// Mitsubishi GX Works2 project: FX3U Rev12-22-jul-2025 1727   PLC: FX3U/FX3UC

PROGRAM 0_HOME
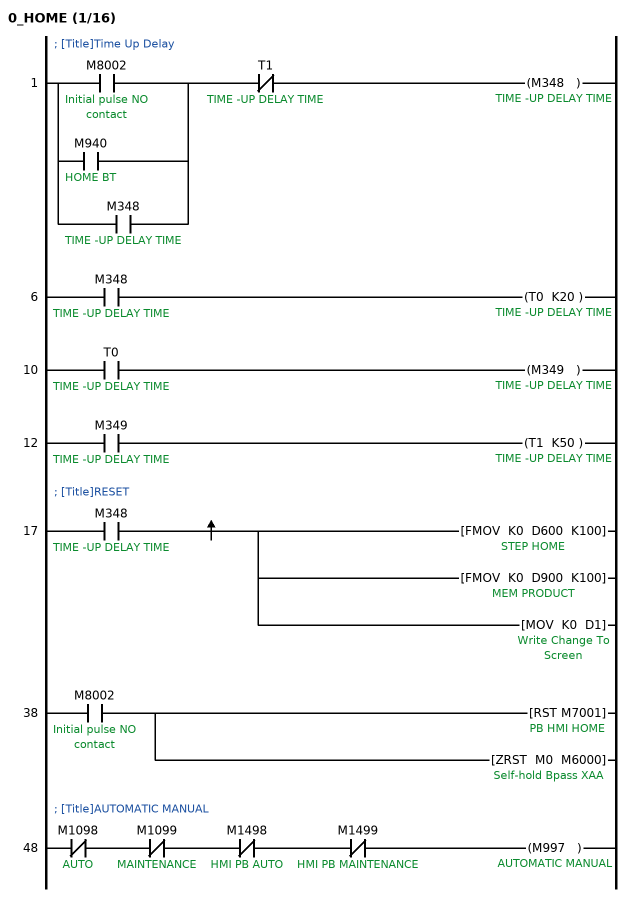
; [Title]Time Up Delay
1     LD      M8002  ; Initial pulse NO contact
      OR      M940  ; HOME BT
      OR      M348  ; TIME -UP DELAY TIME
      ANI     T1  ; TIME -UP DELAY TIME
      OUT     M348  ; TIME -UP DELAY TIME
6     LD      M348  ; TIME -UP DELAY TIME
      OUT     T0 K20  ; TIME -UP DELAY TIME
10    LD      T0  ; TIME -UP DELAY TIME
      OUT     M349  ; TIME -UP DELAY TIME
12    LD      M349  ; TIME -UP DELAY TIME
      OUT     T1 K50  ; TIME -UP DELAY TIME
; [Title]RESET
17    LD      M348  ; TIME -UP DELAY TIME
      MEP
      FMOV    K0 D600 K100  ; STEP HOME
      FMOV    K0 D900 K100  ; MEM PRODUCT
      MOV     K0 D1  ; Write Change To Screen
38    LD      M8002  ; Initial pulse NO contact
      RST     M7001  ; PB HMI HOME
      ZRST    M0 M6000  ; Self-hold Bpass XAA
; [Title]AUTOMATIC MANUAL
48    LDI     M1098  ; AUTO
      ANI     M1099  ; MAINTENANCE
      ANI     M1498  ; HMI PB AUTO
      ANI     M1499  ; HMI PB MAINTENANCE
      OUT     M997  ; AUTOMATIC MANUAL
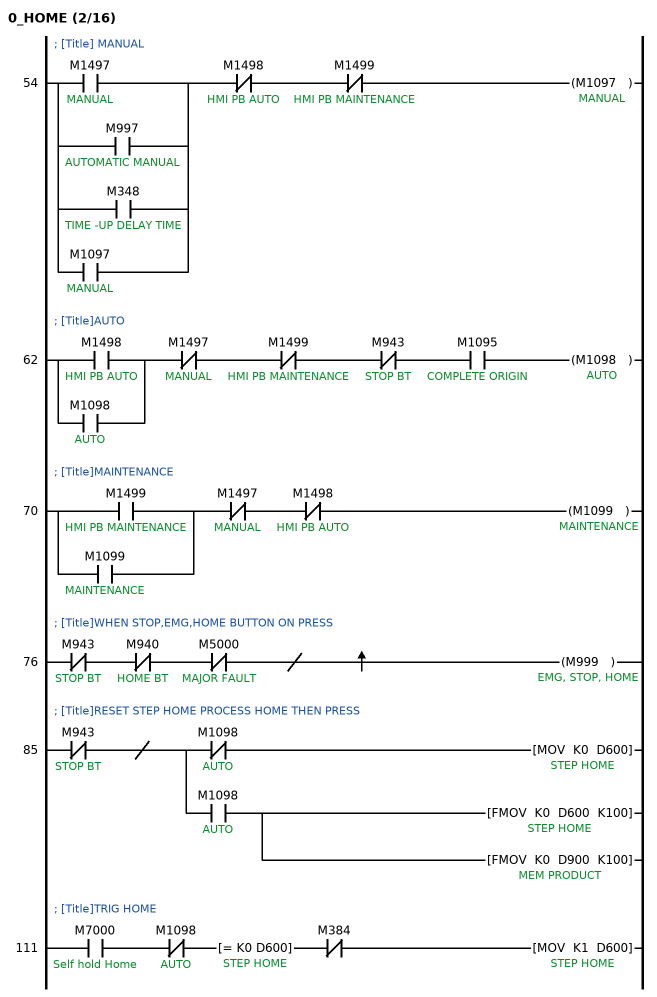
; [Title] MANUAL
54    LD      M1497  ; MANUAL
      OR      M997  ; AUTOMATIC MANUAL
      OR      M348  ; TIME -UP DELAY TIME
      OR      M1097  ; MANUAL
      ANI     M1498  ; HMI PB AUTO
      ANI     M1499  ; HMI PB MAINTENANCE
      OUT     M1097  ; MANUAL
; [Title]AUTO
62    LD      M1498  ; HMI PB AUTO
      OR      M1098  ; AUTO
      ANI     M1497  ; MANUAL
      ANI     M1499  ; HMI PB MAINTENANCE
      ANI     M943  ; STOP BT
      AND     M1095  ; COMPLETE ORIGIN
      OUT     M1098  ; AUTO
; [Title]MAINTENANCE
70    LD      M1499  ; HMI PB MAINTENANCE
      OR      M1099  ; MAINTENANCE
      ANI     M1497  ; MANUAL
      ANI     M1498  ; HMI PB AUTO
      OUT     M1099  ; MAINTENANCE
; [Title]WHEN STOP,EMG,HOME BUTTON ON PRESS
76    LDI     M943  ; STOP BT
      ANI     M940  ; HOME BT
      ANI     M5000  ; MAJOR FAULT
      INV
      MEP
      OUT     M999  ; EMG, STOP, HOME
; [Title]RESET STEP HOME PROCESS HOME THEN PRESS
85    LDI     M943  ; STOP BT
      INV
      MPS
      ANI     M1098  ; AUTO
      MOV     K0 D600
      MPP
      AND     M1098  ; AUTO
      FMOV    K0 D600 K100
      FMOV    K0 D900 K100
; [Title]TRIG HOME
111   LD      M7000  ; Self hold Home
      ANI     M1098  ; AUTO
      AND=    K0 D600  ; STEP HOME
      ANI     M384
      MOV     K1 D600
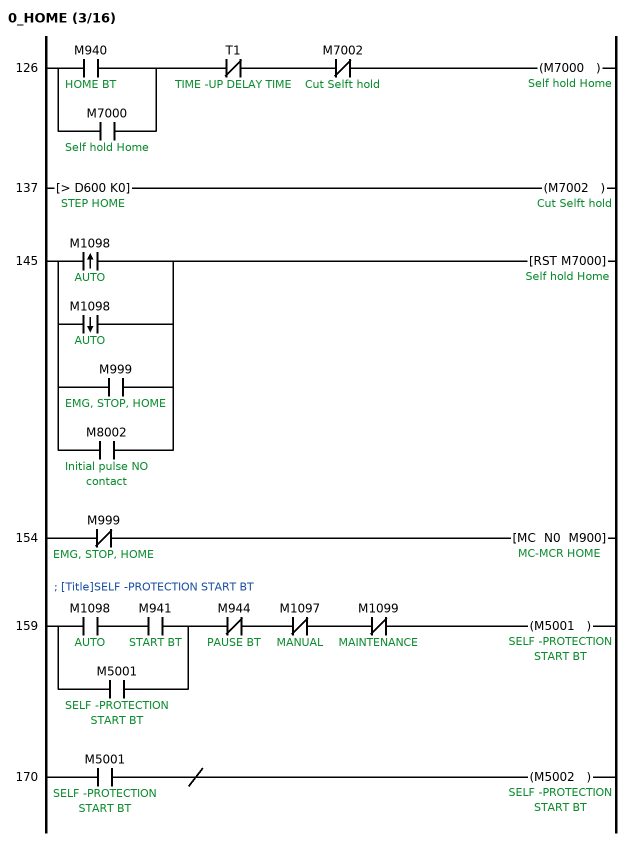
126   LD      M940  ; HOME BT
      OR      M7000  ; Self hold Home
      ANI     T1  ; TIME -UP DELAY TIME
      ANI     M7002  ; Cut Selft hold
      OUT     M7000  ; Self hold Home
137   LD>     D600 K0  ; STEP HOME
      OUT     M7002  ; Cut Selft hold
145   LDP     M1098  ; AUTO
      ORF     M1098  ; AUTO
      OR      M999  ; EMG, STOP, HOME
      OR      M8002  ; Initial pulse NO contact
      RST     M7000  ; Self hold Home
154   LDI     M999  ; EMG, STOP, HOME
      MC      N0 M900  ; MC-MCR HOME
; [Title]SELF -PROTECTION START BT
159   LD      M1098  ; AUTO
      AND     M941  ; START BT
      OR      M5001  ; SELF -PROTECTION START BT
      ANI     M944  ; PAUSE BT
      ANI     M1097  ; MANUAL
      ANI     M1099  ; MAINTENANCE
      OUT     M5001  ; SELF -PROTECTION START BT
170   LD      M5001  ; SELF -PROTECTION START BT
      INV
      OUT     M5002  ; SELF -PROTECTION START BT
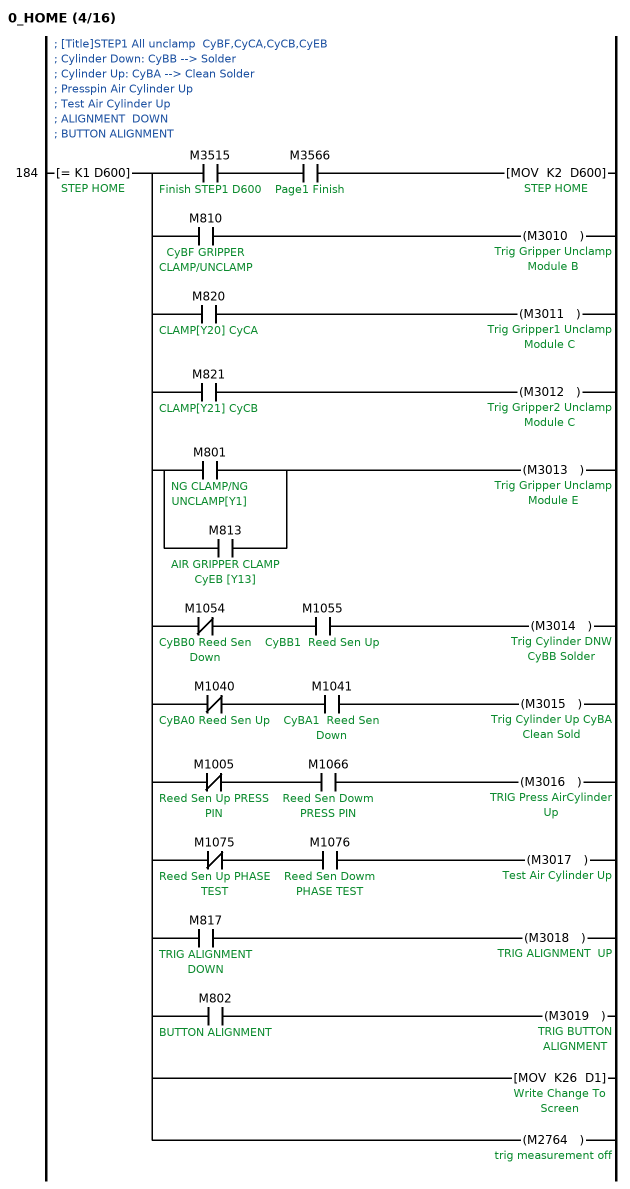
; [Title]STEP1 All unclamp  CyBF,CyCA,CyCB,CyEB
; Cylinder Down: CyBB --> Solder
; Cylinder Up: CyBA --> Clean Solder
; Presspin Air Cylinder Up
; Test Air Cylinder Up
; ALIGNMENT  DOWN
; BUTTON ALIGNMENT
184   LD=     K1 D600  ; STEP HOME
      MPS
      AND     M3515  ; Finish STEP1 D600
      AND     M3566  ; Page1 Finish
      MOV     K2 D600
      MRD
      AND     M810  ; CyBF GRIPPER CLAMP/UNCLAMP
      OUT     M3010  ; Trig Gripper Unclamp Module B
        [note] TRIG Gripper Unclamp Module B
      MRD
      AND     M820  ; CLAMP[Y20] CyCA
      OUT     M3011  ; Trig Gripper1 Unclamp Module C
        [note] TRIG Gripper1 Unclamp Module C
      MRD
      AND     M821  ; CLAMP[Y21] CyCB
      OUT     M3012  ; Trig Gripper2 Unclamp Module C
        [note] TRIG Gripper2 Unclamp Module C
      MRD
      LD      M801  ; NG CLAMP/NG UNCLAMP[Y1]
      OR      M813  ; AIR GRIPPER CLAMP CyEB [Y13]
      ANB
      OUT     M3013  ; Trig Gripper Unclamp Module E
        [note] TRIG Gripper Unclamp Module E
      MRD
      ANI     M1054  ; CyBB0 Reed Sen Down
      AND     M1055  ; CyBB1  Reed Sen Up
      OUT     M3014  ; Trig Cylinder DNW CyBB Solder
        [note] TRIG Cylinder DNW CyBB Solder
      MRD
      ANI     M1040  ; CyBA0 Reed Sen Up
      AND     M1041  ; CyBA1  Reed Sen Down
      OUT     M3015  ; Trig Cylinder Up CyBA Clean Sold
        [note] TRIG Cylinder Up CyBA Clean
      MRD
      ANI     M1005  ; Reed Sen Up PRESS PIN
      AND     M1066  ; Reed Sen Dowm PRESS PIN
      OUT     M3016  ; TRIG Press AirCylinder Up
        [note] TRIG Press AirCylinder Up
      MRD
      ANI     M1075  ; Reed Sen Up PHASE TEST
      AND     M1076  ; Reed Sen Dowm PHASE TEST
      OUT     M3017  ; Test Air Cylinder Up
        [note] TRIG Test Air Cylinder Up
      MRD
      AND     M817  ; TRIG ALIGNMENT  DOWN
      OUT     M3018  ; TRIG ALIGNMENT  UP
        [note] TRIG ALIGNMENT  UP
      MRD
      AND     M802  ; BUTTON ALIGNMENT
      OUT     M3019  ; TRIG BUTTON ALIGNMENT
        [note] TRIG BUTTON ALIGNMENT
      MPP
      MOV     K26 D1
      OUT     M2764  ; trig measurement off
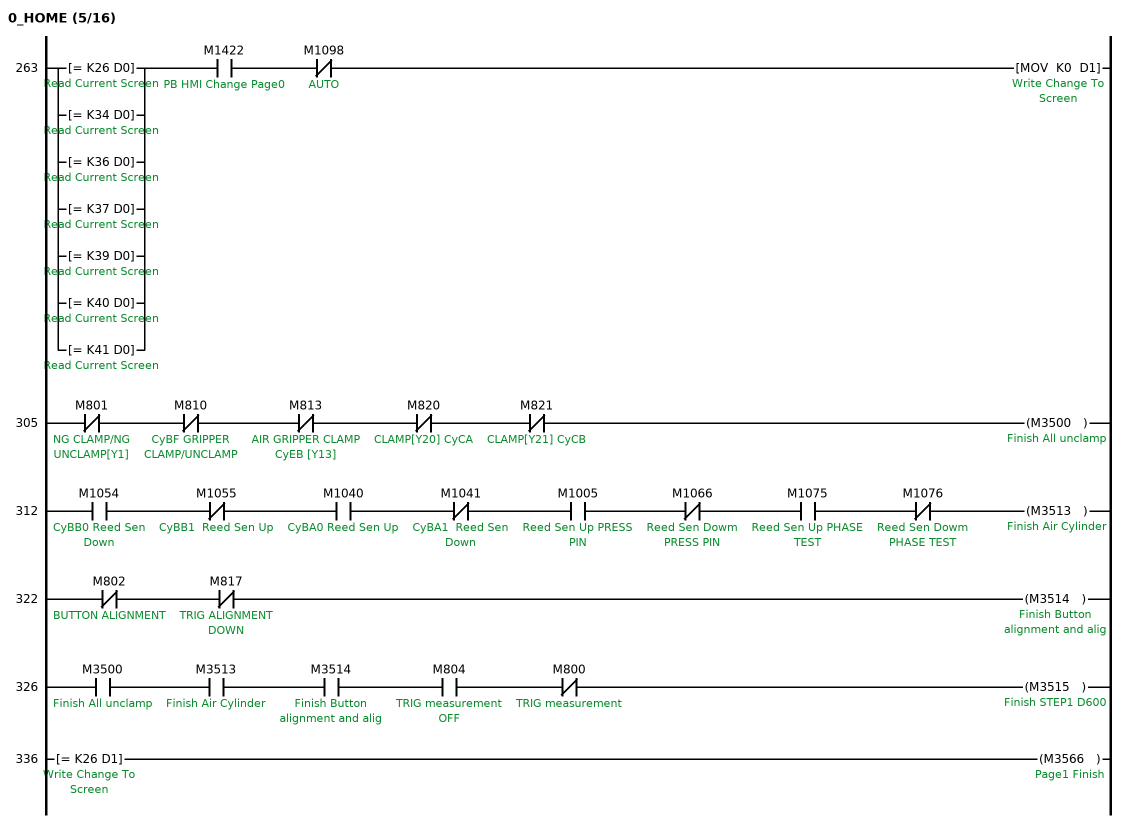
263   LD=     K26 D0  ; Read Current Screen
      OR=     K34 D0  ; Read Current Screen
      OR=     K36 D0  ; Read Current Screen
      OR=     K37 D0  ; Read Current Screen
      OR=     K39 D0  ; Read Current Screen
      OR=     K40 D0  ; Read Current Screen
      OR=     K41 D0  ; Read Current Screen
      AND     M1422  ; PB HMI Change Page0
      ANI     M1098  ; AUTO
      MOV     K0 D1
305   LDI     M801  ; NG CLAMP/NG UNCLAMP[Y1]
      ANI     M810  ; CyBF GRIPPER CLAMP/UNCLAMP
      ANI     M813  ; AIR GRIPPER CLAMP CyEB [Y13]
      ANI     M820  ; CLAMP[Y20] CyCA
      ANI     M821  ; CLAMP[Y21] CyCB
      OUT     M3500  ; Finish All unclamp
312   LD      M1054  ; CyBB0 Reed Sen Down
      ANI     M1055  ; CyBB1  Reed Sen Up
      AND     M1040  ; CyBA0 Reed Sen Up
      ANI     M1041  ; CyBA1  Reed Sen Down
      AND     M1005  ; Reed Sen Up PRESS PIN
      ANI     M1066  ; Reed Sen Dowm PRESS PIN
      AND     M1075  ; Reed Sen Up PHASE TEST
      ANI     M1076  ; Reed Sen Dowm PHASE TEST
      OUT     M3513  ; Finish Air Cylinder
322   LDI     M802  ; BUTTON ALIGNMENT
      ANI     M817  ; TRIG ALIGNMENT  DOWN
      OUT     M3514  ; Finish Button alignment and alig
326   LD      M3500  ; Finish All unclamp
      AND     M3513  ; Finish Air Cylinder
      AND     M3514  ; Finish Button alignment and alig
      AND     M804  ; TRIG measurement OFF
      ANI     M800  ; TRIG measurement
      OUT     M3515  ; Finish STEP1 D600
336   LD=     K26 D1  ; Write Change To Screen
      OUT     M3566  ; Page1 Finish
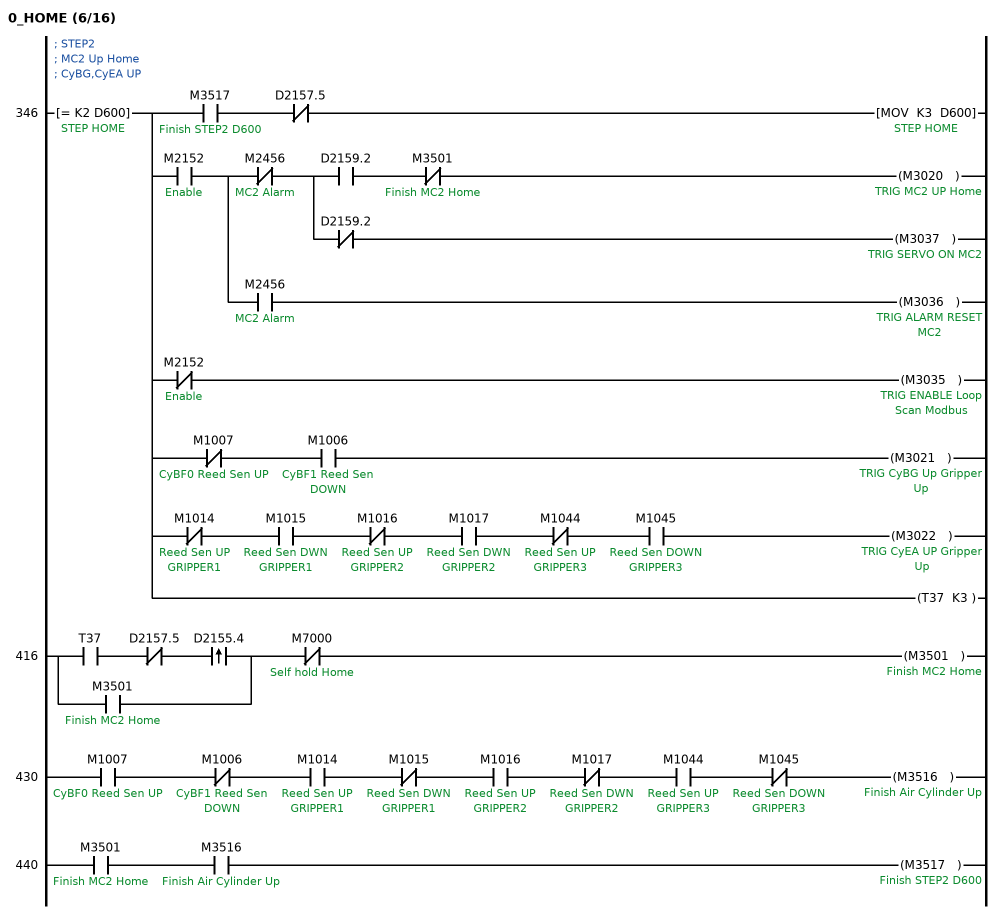
; STEP2
; MC2 Up Home
; CyBG,CyEA UP
346   LD=     K2 D600  ; STEP HOME
      MPS
      AND     M3517  ; Finish STEP2 D600
      ANI     D2157.5
      MOV     K3 D600
      MRD
      AND     M2152  ; Enable
      MPS
      ANI     M2456  ; MC2 Alarm
      MPS
      AND     D2159.2
      ANI     M3501  ; Finish MC2 Home
      OUT     M3020  ; TRIG MC2 UP Home
        [note] TRIG MC2 UP Home
      MPP
      ANI     D2159.2
      OUT     M3037  ; TRIG SERVO ON MC2
        [note] TRIG SERVO ON MC2
      MPP
      AND     M2456  ; MC2 Alarm
      OUT     M3036  ; TRIG ALARM RESET MC2
        [note] TRIG ALARM RESET MC2
      MRD
      ANI     M2152  ; Enable
      OUT     M3035  ; TRIG ENABLE Loop Scan Modbus
        [note] TRIG ENABLE Loop Scan Modbus
      MRD
      ANI     M1007  ; CyBF0 Reed Sen UP
      AND     M1006  ; CyBF1 Reed Sen DOWN
      OUT     M3021  ; TRIG CyBG Up Gripper Up
        [note] TRIG CyBG Up Gripper Up
      MRD
      ANI     M1014  ; Reed Sen UP GRIPPER1
      AND     M1015  ; Reed Sen DWN GRIPPER1
      ANI     M1016  ; Reed Sen UP GRIPPER2
      AND     M1017  ; Reed Sen DWN GRIPPER2
      ANI     M1044  ; Reed Sen UP GRIPPER3
      AND     M1045  ; Reed Sen DOWN GRIPPER3
      OUT     M3022  ; TRIG CyEA UP Gripper Up
        [note] TRIG CyEA UP Gripper Up
      MPP
      OUT     T37 K3
416   LD      T37
      ANI     D2157.5
      ANDP    D2155.4
      OR      M3501  ; Finish MC2 Home
      ANI     M7000  ; Self hold Home
      OUT     M3501  ; Finish MC2 Home
430   LD      M1007  ; CyBF0 Reed Sen UP
      ANI     M1006  ; CyBF1 Reed Sen DOWN
      AND     M1014  ; Reed Sen UP GRIPPER1
      ANI     M1015  ; Reed Sen DWN GRIPPER1
      AND     M1016  ; Reed Sen UP GRIPPER2
      ANI     M1017  ; Reed Sen DWN GRIPPER2
      AND     M1044  ; Reed Sen UP GRIPPER3
      ANI     M1045  ; Reed Sen DOWN GRIPPER3
      OUT     M3516  ; Finish Air Cylinder Up
440   LD      M3501  ; Finish MC2 Home
      AND     M3516  ; Finish Air Cylinder Up
      OUT     M3517  ; Finish STEP2 D600
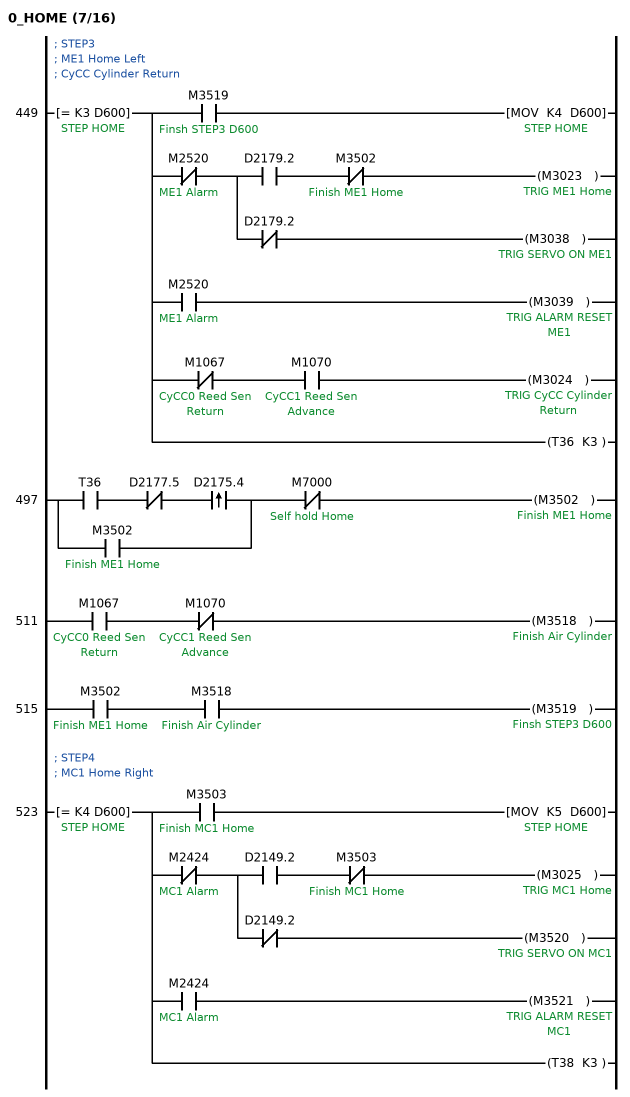
; STEP3
; ME1 Home Left
; CyCC Cylinder Return
449   LD=     K3 D600  ; STEP HOME
      MPS
      AND     M3519  ; Finsh STEP3 D600
      MOV     K4 D600
      MRD
      ANI     M2520  ; ME1 Alarm
      MPS
      AND     D2179.2
      ANI     M3502  ; Finish ME1 Home
      OUT     M3023  ; TRIG ME1 Home
        [note] TRIG ME1 Home
      MPP
      ANI     D2179.2
      OUT     M3038  ; TRIG SERVO ON ME1
        [note] TRIG SERVO ON ME1
      MRD
      AND     M2520  ; ME1 Alarm
      OUT     M3039  ; TRIG ALARM RESET ME1
        [note] TRIG ALARM RESET ME1
      MRD
      ANI     M1067  ; CyCC0 Reed Sen Return
      AND     M1070  ; CyCC1 Reed Sen  Advance
      OUT     M3024  ; TRIG CyCC Cylinder Return
        [note] TRIG CyCC Cylinder Return
      MPP
      OUT     T36 K3
497   LD      T36
      ANI     D2177.5
      ANDP    D2175.4
      OR      M3502  ; Finish ME1 Home
      ANI     M7000  ; Self hold Home
      OUT     M3502  ; Finish ME1 Home
511   LD      M1067  ; CyCC0 Reed Sen Return
      ANI     M1070  ; CyCC1 Reed Sen  Advance
      OUT     M3518  ; Finish Air Cylinder
515   LD      M3502  ; Finish ME1 Home
      AND     M3518  ; Finish Air Cylinder
      OUT     M3519  ; Finsh STEP3 D600
; STEP4
; MC1 Home Right
523   LD=     K4 D600  ; STEP HOME
      MPS
      AND     M3503  ; Finish MC1 Home
      MOV     K5 D600
      MRD
      ANI     M2424  ; MC1 Alarm
      MPS
      AND     D2149.2
      ANI     M3503  ; Finish MC1 Home
      OUT     M3025  ; TRIG MC1 Home
        [note] TRIG MC1 Home
      MPP
      ANI     D2149.2
      OUT     M3520  ; TRIG SERVO ON MC1
        [note] TRIG SERVO ON MC1
      MRD
      AND     M2424  ; MC1 Alarm
      OUT     M3521  ; TRIG ALARM RESET MC1
        [note] TRIG ALARM RESET MC1
      MPP
      OUT     T38 K3
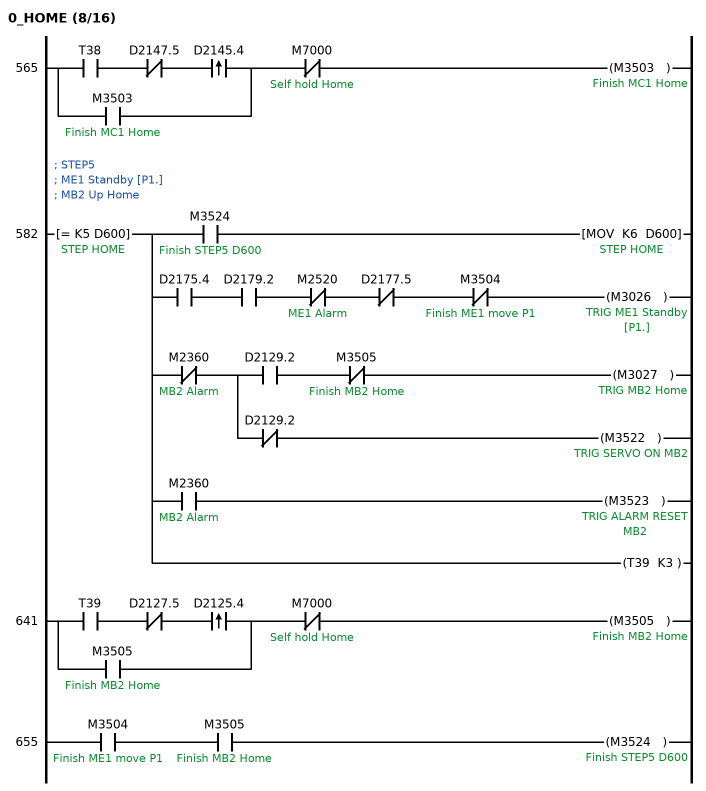
565   LD      T38
      ANI     D2147.5
      ANDP    D2145.4
      OR      M3503  ; Finish MC1 Home
      ANI     M7000  ; Self hold Home
      OUT     M3503  ; Finish MC1 Home
; STEP5
; ME1 Standby [P1.]
; MB2 Up Home
582   LD=     K5 D600  ; STEP HOME
      MPS
      AND     M3524  ; Finish STEP5 D600
      MOV     K6 D600
      MRD
      AND     D2175.4
      AND     D2179.2
      ANI     M2520  ; ME1 Alarm
      ANI     D2177.5
      ANI     M3504  ; Finish ME1 move P1
      OUT     M3026  ; TRIG ME1 Standby [P1.]
        [note] ME1 Standby [P1.]
      MRD
      ANI     M2360  ; MB2 Alarm
      MPS
      AND     D2129.2
      ANI     M3505  ; Finish MB2 Home
      OUT     M3027  ; TRIG MB2 Home
        [note] TRIG MB2 Home
      MPP
      ANI     D2129.2
      OUT     M3522  ; TRIG SERVO ON MB2
        [note] TRIG SERVO ON MB2
      MRD
      AND     M2360  ; MB2 Alarm
      OUT     M3523  ; TRIG ALARM RESET MB2
        [note] TRIG ALARM RESET MB2
      MPP
      OUT     T39 K3
641   LD      T39
      ANI     D2127.5
      ANDP    D2125.4
      OR      M3505  ; Finish MB2 Home
      ANI     M7000  ; Self hold Home
      OUT     M3505  ; Finish MB2 Home
655   LD      M3504  ; Finish ME1 move P1
      AND     M3505  ; Finish MB2 Home
      OUT     M3524  ; Finish STEP5 D600
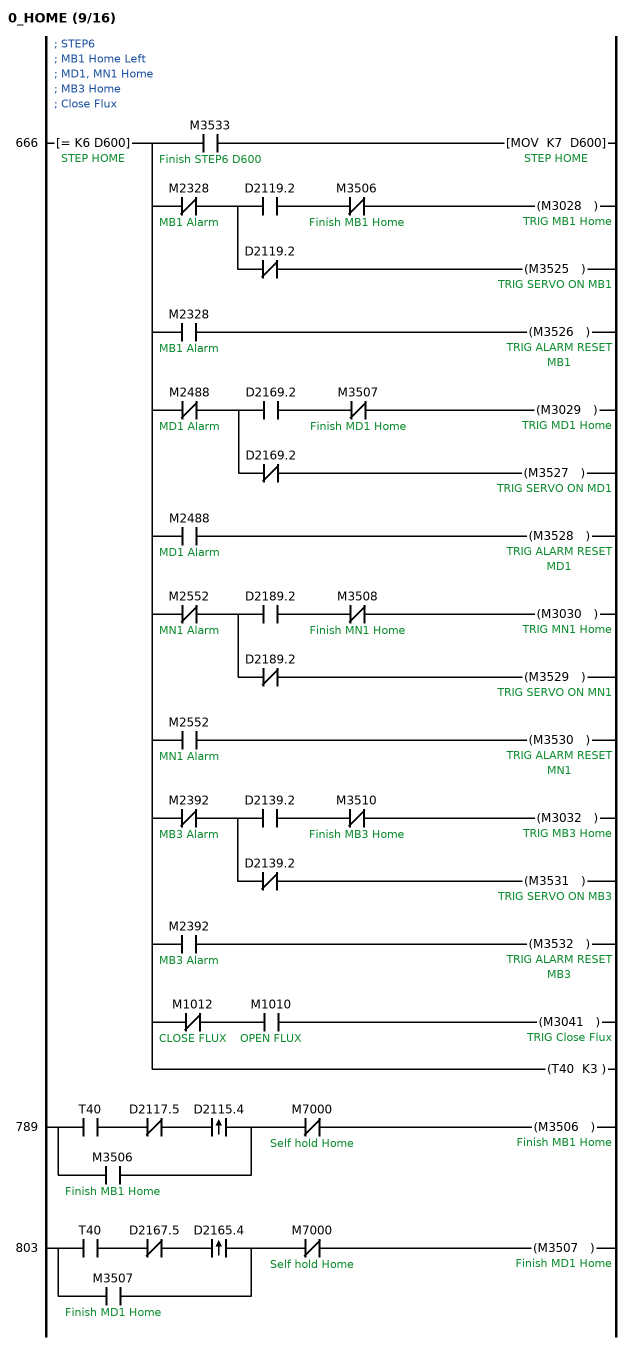
; STEP6
; MB1 Home Left
; MD1, MN1 Home
; MB3 Home
; Close Flux
666   LD=     K6 D600  ; STEP HOME
      MPS
      AND     M3533  ; Finish STEP6 D600
      MOV     K7 D600
      MRD
      ANI     M2328  ; MB1 Alarm
      MPS
      AND     D2119.2
      ANI     M3506  ; Finish MB1 Home
      OUT     M3028  ; TRIG MB1 Home
        [note] TRIG MB1 Home
      MPP
      ANI     D2119.2
      OUT     M3525  ; TRIG SERVO ON MB1
        [note] TRIG SERVO ON MB1
      MRD
      AND     M2328  ; MB1 Alarm
      OUT     M3526  ; TRIG ALARM RESET MB1
        [note] TRIG ALARM RESET MB1
      MRD
      ANI     M2488  ; MD1 Alarm
      MPS
      AND     D2169.2
      ANI     M3507  ; Finish MD1 Home
      OUT     M3029  ; TRIG MD1 Home
        [note] TRIG MD1 Home
      MPP
      ANI     D2169.2
      OUT     M3527  ; TRIG SERVO ON MD1
        [note] TRIG SERVO ON MD1
      MRD
      AND     M2488  ; MD1 Alarm
      OUT     M3528  ; TRIG ALARM RESET MD1
        [note] TRIG ALARM RESET MD1
      MRD
      ANI     M2552  ; MN1 Alarm
      MPS
      AND     D2189.2
      ANI     M3508  ; Finish MN1 Home
      OUT     M3030  ; TRIG MN1 Home
        [note] TRIG MN1 Home
      MPP
      ANI     D2189.2
      OUT     M3529  ; TRIG SERVO ON MN1
        [note] TRIG SERVO ON MN1
      MRD
      AND     M2552  ; MN1 Alarm
      OUT     M3530  ; TRIG ALARM RESET MN1
        [note] TRIG ALARM RESET MN1
      MRD
      ANI     M2392  ; MB3 Alarm
      MPS
      AND     D2139.2
      ANI     M3510  ; Finish MB3 Home
      OUT     M3032  ; TRIG MB3 Home
        [note] TRIG MB3 Home
      MPP
      ANI     D2139.2
      OUT     M3531  ; TRIG SERVO ON MB3
        [note] TRIG SERVO ON MB3
      MRD
      AND     M2392  ; MB3 Alarm
      OUT     M3532  ; TRIG ALARM RESET MB3
        [note] TRIG ALARM RESET MB3
      MRD
      ANI     M1012  ; CLOSE FLUX
      AND     M1010  ; OPEN FLUX
      OUT     M3041  ; TRIG Close Flux
        [note] TRIG Close Flux
      MPP
      OUT     T40 K3
789   LD      T40
      ANI     D2117.5
      ANDP    D2115.4
      OR      M3506  ; Finish MB1 Home
      ANI     M7000  ; Self hold Home
      OUT     M3506  ; Finish MB1 Home
803   LD      T40
      ANI     D2167.5
      ANDP    D2165.4
      OR      M3507  ; Finish MD1 Home
      ANI     M7000  ; Self hold Home
      OUT     M3507  ; Finish MD1 Home
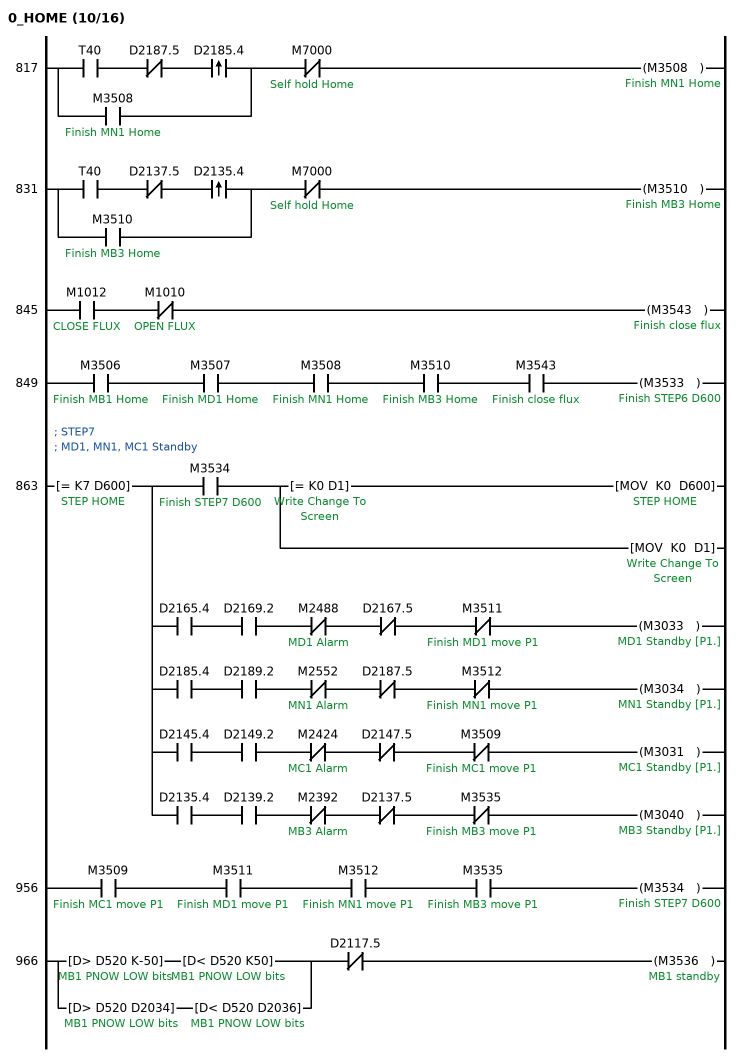
817   LD      T40
      ANI     D2187.5
      ANDP    D2185.4
      OR      M3508  ; Finish MN1 Home
      ANI     M7000  ; Self hold Home
      OUT     M3508  ; Finish MN1 Home
831   LD      T40
      ANI     D2137.5
      ANDP    D2135.4
      OR      M3510  ; Finish MB3 Home
      ANI     M7000  ; Self hold Home
      OUT     M3510  ; Finish MB3 Home
845   LD      M1012  ; CLOSE FLUX
      ANI     M1010  ; OPEN FLUX
      OUT     M3543  ; Finish close flux
849   LD      M3506  ; Finish MB1 Home
      AND     M3507  ; Finish MD1 Home
      AND     M3508  ; Finish MN1 Home
      AND     M3510  ; Finish MB3 Home
      AND     M3543  ; Finish close flux
      OUT     M3533  ; Finish STEP6 D600
; STEP7
; MD1, MN1, MC1 Standby
863   LD=     K7 D600  ; STEP HOME
      MPS
      AND     M3534  ; Finish STEP7 D600
      MPS
      AND=    K0 D1  ; Write Change To Screen
      MOV     K0 D600
      MPP
      MOV     K0 D1
      MRD
      AND     D2165.4
      AND     D2169.2
      ANI     M2488  ; MD1 Alarm
      ANI     D2167.5
      ANI     M3511  ; Finish MD1 move P1
      OUT     M3033  ; MD1 Standby [P1.]
        [note] MD1 Standby [P1.]
      MRD
      AND     D2185.4
      AND     D2189.2
      ANI     M2552  ; MN1 Alarm
      ANI     D2187.5
      ANI     M3512  ; Finish MN1 move P1
      OUT     M3034  ; MN1 Standby [P1.]
        [note] MN1 Standby [P1.]
      MRD
      AND     D2145.4
      AND     D2149.2
      ANI     M2424  ; MC1 Alarm
      ANI     D2147.5
      ANI     M3509  ; Finish MC1 move P1
      OUT     M3031  ; MC1 Standby [P1.]
        [note] MC1 Standby [P1.]
      MPP
      AND     D2135.4
      AND     D2139.2
      ANI     M2392  ; MB3 Alarm
      ANI     D2137.5
      ANI     M3535  ; Finish MB3 move P1
      OUT     M3040  ; MB3 Standby [P1.]
        [note] MB3 Standby [P1.]
956   LD      M3509  ; Finish MC1 move P1
      AND     M3511  ; Finish MD1 move P1
      AND     M3512  ; Finish MN1 move P1
      AND     M3535  ; Finish MB3 move P1
      OUT     M3534  ; Finish STEP7 D600
966   LDD>    D520 K-50  ; MB1 PNOW LOW bits
      ANDD<   D520 K50  ; MB1 PNOW LOW bits
      LDD>    D520 D2034  ; MB1 PNOW LOW bits
      ANDD<   D520 D2036  ; MB1 PNOW LOW bits
      ORB
      ANI     D2117.5
      OUT     M3536  ; MB1 standby
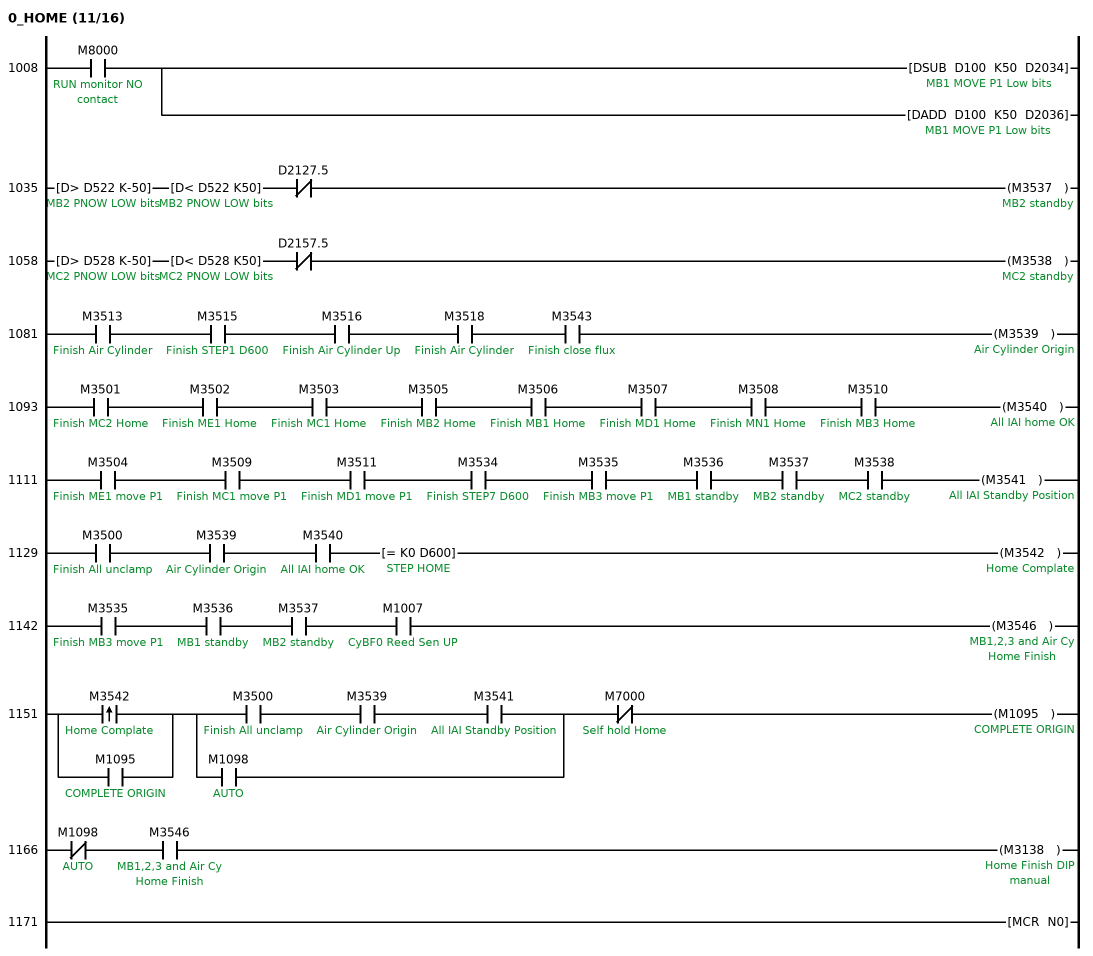
1008  LD      M8000  ; RUN monitor NO contact
      DSUB    D100 K50 D2034  ; MB1 MOVE P1 Low bits
      DADD    D100 K50 D2036
1035  LDD>    D522 K-50  ; MB2 PNOW LOW bits
      ANDD<   D522 K50  ; MB2 PNOW LOW bits
      ANI     D2127.5
      OUT     M3537  ; MB2 standby
1058  LDD>    D528 K-50  ; MC2 PNOW LOW bits
      ANDD<   D528 K50  ; MC2 PNOW LOW bits
      ANI     D2157.5
      OUT     M3538  ; MC2 standby
1081  LD      M3513  ; Finish Air Cylinder
      AND     M3515  ; Finish STEP1 D600
      AND     M3516  ; Finish Air Cylinder Up
      AND     M3518  ; Finish Air Cylinder
      AND     M3543  ; Finish close flux
      OUT     M3539  ; Air Cylinder Origin
1093  LD      M3501  ; Finish MC2 Home
      AND     M3502  ; Finish ME1 Home
      AND     M3503  ; Finish MC1 Home
      AND     M3505  ; Finish MB2 Home
      AND     M3506  ; Finish MB1 Home
      AND     M3507  ; Finish MD1 Home
      AND     M3508  ; Finish MN1 Home
      AND     M3510  ; Finish MB3 Home
      OUT     M3540  ; All IAI home OK
1111  LD      M3504  ; Finish ME1 move P1
      AND     M3509  ; Finish MC1 move P1
      AND     M3511  ; Finish MD1 move P1
      AND     M3534  ; Finish STEP7 D600
      AND     M3535  ; Finish MB3 move P1
      AND     M3536  ; MB1 standby
      AND     M3537  ; MB2 standby
      AND     M3538  ; MC2 standby
      OUT     M3541  ; All IAI Standby Position
1129  LD      M3500  ; Finish All unclamp
      AND     M3539  ; Air Cylinder Origin
      AND     M3540  ; All IAI home OK
      AND=    K0 D600  ; STEP HOME
      OUT     M3542  ; Home Complate
1142  LD      M3535  ; Finish MB3 move P1
      AND     M3536  ; MB1 standby
      AND     M3537  ; MB2 standby
      AND     M1007  ; CyBF0 Reed Sen UP
      OUT     M3546  ; MB1,2,3 and Air Cy Home Finish
1151  LDP     M3542  ; Home Complate
      OR      M1095  ; COMPLETE ORIGIN
      LD      M3500  ; Finish All unclamp
      AND     M3539  ; Air Cylinder Origin
      AND     M3541  ; All IAI Standby Position
      OR      M1098  ; AUTO
      ANB
      ANI     M7000  ; Self hold Home
      OUT     M1095  ; COMPLETE ORIGIN
1166  LDI     M1098  ; AUTO
      AND     M3546  ; MB1,2,3 and Air Cy Home Finish
      OUT     M3138  ; Home Finish DIP manual
1171  MCR     N0
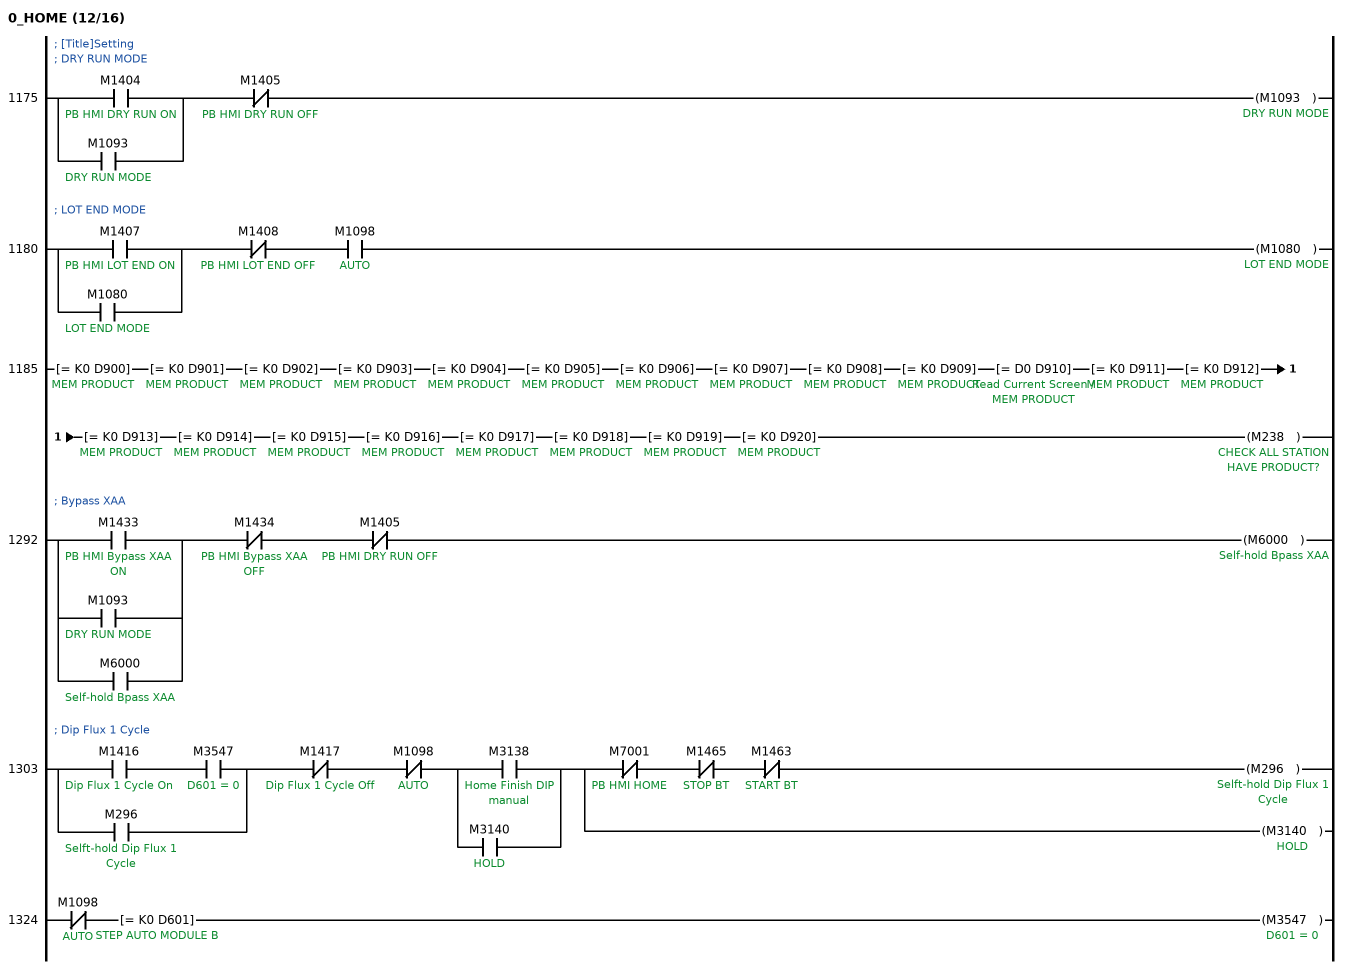
; [Title]Setting
; DRY RUN MODE
1175  LD      M1404  ; PB HMI DRY RUN ON
      OR      M1093  ; DRY RUN MODE
      ANI     M1405  ; PB HMI DRY RUN OFF
      OUT     M1093  ; DRY RUN MODE
; LOT END MODE
1180  LD      M1407  ; PB HMI LOT END ON
      OR      M1080  ; LOT END MODE
      ANI     M1408  ; PB HMI LOT END OFF
      AND     M1098  ; AUTO
      OUT     M1080  ; LOT END MODE
1185  LD=     K0 D900  ; MEM PRODUCT
      AND=    K0 D901  ; MEM PRODUCT
      AND=    K0 D902  ; MEM PRODUCT
      AND=    K0 D903  ; MEM PRODUCT
      AND=    K0 D904  ; MEM PRODUCT
      AND=    K0 D905  ; MEM PRODUCT
      AND=    K0 D906  ; MEM PRODUCT
      AND=    K0 D907  ; MEM PRODUCT
      AND=    K0 D908  ; MEM PRODUCT
      AND=    K0 D909  ; MEM PRODUCT
      AND=    D0 D910  ; Read Current Screen / MEM PRODUCT
      AND=    K0 D911  ; MEM PRODUCT
      AND=    K0 D912  ; MEM PRODUCT
      AND=    K0 D913  ; MEM PRODUCT
      AND=    K0 D914  ; MEM PRODUCT
      AND=    K0 D915  ; MEM PRODUCT
      AND=    K0 D916  ; MEM PRODUCT
      AND=    K0 D917  ; MEM PRODUCT
      AND=    K0 D918  ; MEM PRODUCT
      AND=    K0 D919  ; MEM PRODUCT
      AND=    K0 D920  ; MEM PRODUCT
      OUT     M238  ; CHECK ALL STATION HAVE PRODUCT?
; Bypass XAA
1292  LD      M1433  ; PB HMI Bypass XAA ON
      OR      M1093  ; DRY RUN MODE
      OR      M6000  ; Self-hold Bpass XAA
      ANI     M1434  ; PB HMI Bypass XAA OFF
      ANI     M1405  ; PB HMI DRY RUN OFF
      OUT     M6000  ; Self-hold Bpass XAA
; Dip Flux 1 Cycle
1303  LD      M1416  ; Dip Flux 1 Cycle On
      AND     M3547  ; D601 = 0
      OR      M296  ; Selft-hold Dip Flux 1 Cycle
      ANI     M1417  ; Dip Flux 1 Cycle Off
      ANI     M1098  ; AUTO
      LD      M3138  ; Home Finish DIP manual
      OR      M3140  ; HOLD
      ANB
      MPS
      ANI     M7001  ; PB HMI HOME
      ANI     M1465  ; STOP BT
      ANI     M1463  ; START BT
      OUT     M296  ; Selft-hold Dip Flux 1 Cycle
      MPP
      OUT     M3140  ; HOLD
1324  LDI     M1098  ; AUTO
      AND=    K0 D601  ; STEP AUTO MODULE B
      OUT     M3547  ; D601 = 0
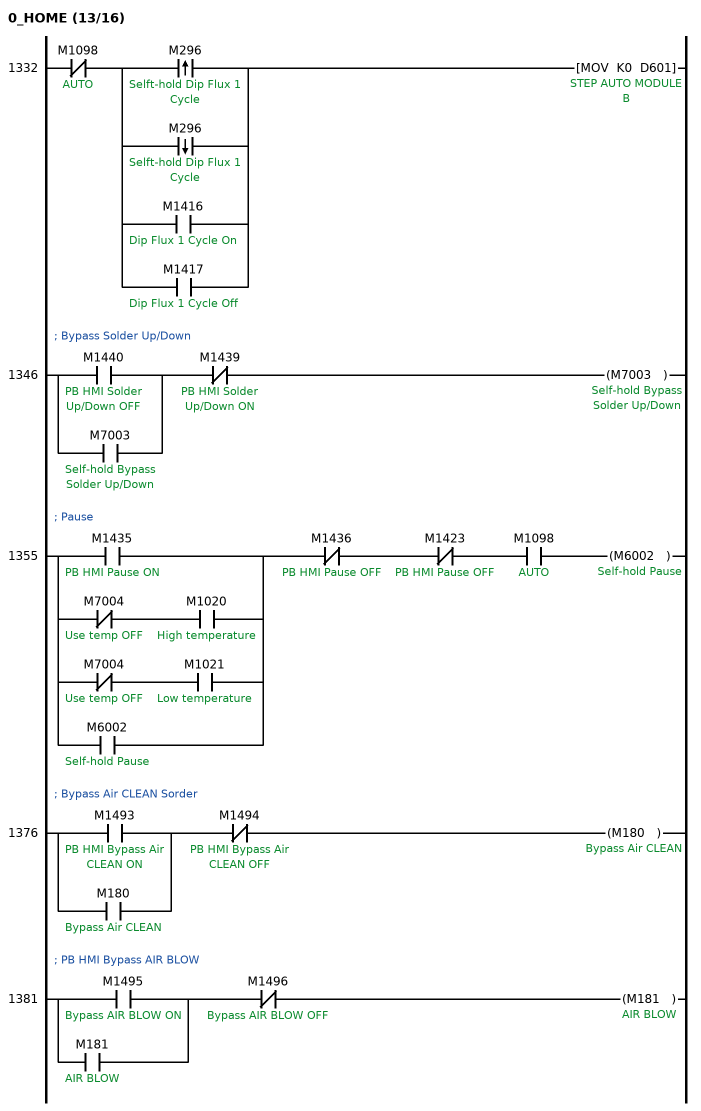
1332  LDI     M1098  ; AUTO
      LDP     M296  ; Selft-hold Dip Flux 1 Cycle
      ORF     M296  ; Selft-hold Dip Flux 1 Cycle
      OR      M1416  ; Dip Flux 1 Cycle On
      OR      M1417  ; Dip Flux 1 Cycle Off
      ANB
      MOV     K0 D601
; Bypass Solder Up/Down
1346  LD      M1440  ; PB HMI Solder Up/Down OFF
      OR      M7003  ; Self-hold Bypass Solder Up/Down
      ANI     M1439  ; PB HMI Solder Up/Down ON
      OUT     M7003  ; Self-hold Bypass Solder Up/Down
; Pause
1355  LD      M1435  ; PB HMI Pause ON
      LDI     M7004  ; Use temp OFF
      AND     M1020  ; High temperature
      ORB
      LDI     M7004  ; Use temp OFF
      AND     M1021  ; Low temperature
      ORB
      OR      M6002  ; Self-hold Pause
      ANI     M1436  ; PB HMI Pause OFF
      ANI     M1423  ; PB HMI Pause OFF
      AND     M1098  ; AUTO
      OUT     M6002  ; Self-hold Pause
; Bypass Air CLEAN Sorder
1376  LD      M1493  ; PB HMI Bypass Air CLEAN ON
      OR      M180  ; Bypass Air CLEAN
      ANI     M1494  ; PB HMI Bypass Air CLEAN OFF
      OUT     M180  ; Bypass Air CLEAN
; PB HMI Bypass AIR BLOW
1381  LD      M1495  ; Bypass AIR BLOW ON
      OR      M181  ; AIR BLOW
      ANI     M1496  ; Bypass AIR BLOW OFF
      OUT     M181  ; AIR BLOW
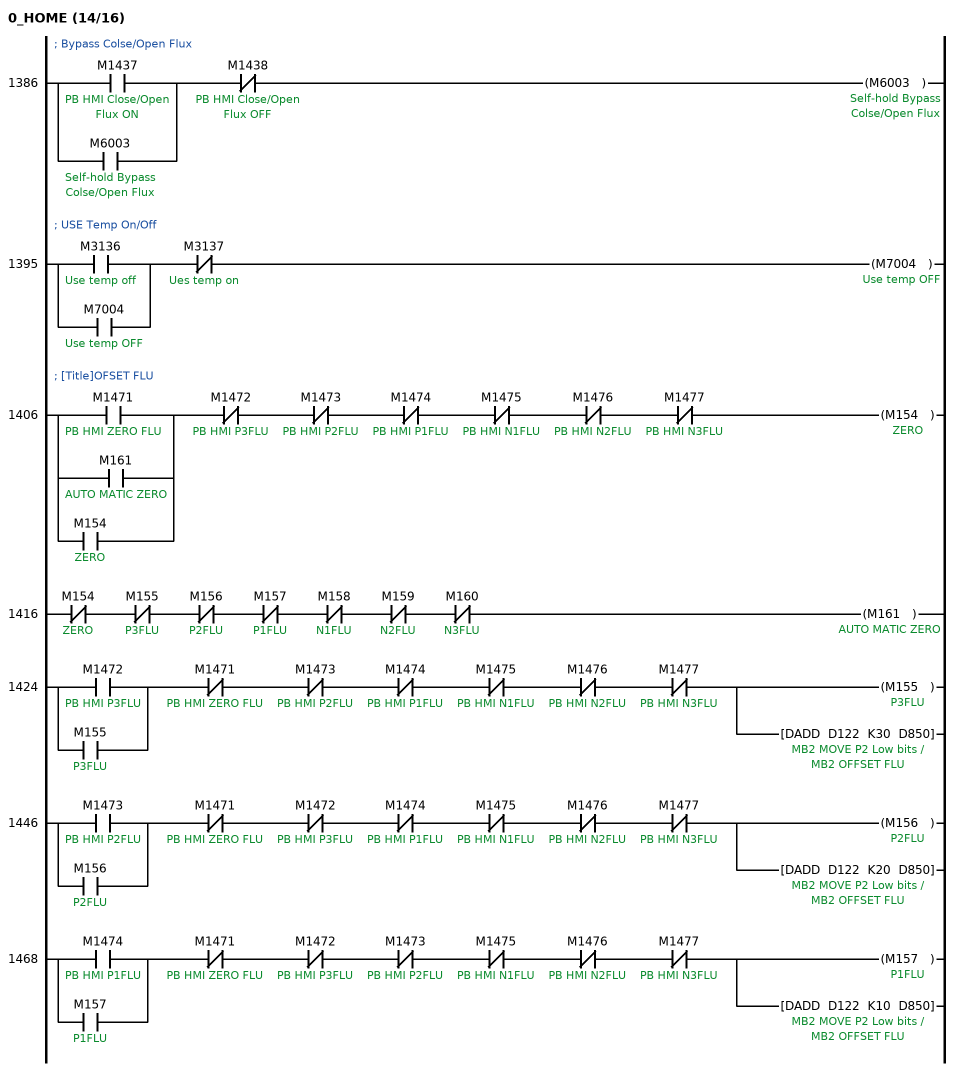
; Bypass Colse/Open Flux
1386  LD      M1437  ; PB HMI Close/Open Flux ON
      OR      M6003  ; Self-hold Bypass Colse/Open Flux
      ANI     M1438  ; PB HMI Close/Open Flux OFF
      OUT     M6003  ; Self-hold Bypass Colse/Open Flux
; USE Temp On/Off
1395  LD      M3136  ; Use temp off
      OR      M7004  ; Use temp OFF
      ANI     M3137  ; Ues temp on
      OUT     M7004  ; Use temp OFF
; [Title]OFSET FLU
1406  LD      M1471  ; PB HMI ZERO FLU
      OR      M161  ; AUTO MATIC ZERO
      OR      M154  ; ZERO
      ANI     M1472  ; PB HMI P3FLU
      ANI     M1473  ; PB HMI P2FLU
      ANI     M1474  ; PB HMI P1FLU
      ANI     M1475  ; PB HMI N1FLU
      ANI     M1476  ; PB HMI N2FLU
      ANI     M1477  ; PB HMI N3FLU
      OUT     M154  ; ZERO
1416  LDI     M154  ; ZERO
      ANI     M155  ; P3FLU
      ANI     M156  ; P2FLU
      ANI     M157  ; P1FLU
      ANI     M158  ; N1FLU
      ANI     M159  ; N2FLU
      ANI     M160  ; N3FLU
      OUT     M161  ; AUTO MATIC ZERO
1424  LD      M1472  ; PB HMI P3FLU
      OR      M155  ; P3FLU
      ANI     M1471  ; PB HMI ZERO FLU
      ANI     M1473  ; PB HMI P2FLU
      ANI     M1474  ; PB HMI P1FLU
      ANI     M1475  ; PB HMI N1FLU
      ANI     M1476  ; PB HMI N2FLU
      ANI     M1477  ; PB HMI N3FLU
      OUT     M155  ; P3FLU
      DADD    D122 K30 D850  ; MB2 MOVE P2 Low bits / MB2 OFFSET FLU
1446  LD      M1473  ; PB HMI P2FLU
      OR      M156  ; P2FLU
      ANI     M1471  ; PB HMI ZERO FLU
      ANI     M1472  ; PB HMI P3FLU
      ANI     M1474  ; PB HMI P1FLU
      ANI     M1475  ; PB HMI N1FLU
      ANI     M1476  ; PB HMI N2FLU
      ANI     M1477  ; PB HMI N3FLU
      OUT     M156  ; P2FLU
      DADD    D122 K20 D850
1468  LD      M1474  ; PB HMI P1FLU
      OR      M157  ; P1FLU
      ANI     M1471  ; PB HMI ZERO FLU
      ANI     M1472  ; PB HMI P3FLU
      ANI     M1473  ; PB HMI P2FLU
      ANI     M1475  ; PB HMI N1FLU
      ANI     M1476  ; PB HMI N2FLU
      ANI     M1477  ; PB HMI N3FLU
      OUT     M157  ; P1FLU
      DADD    D122 K10 D850
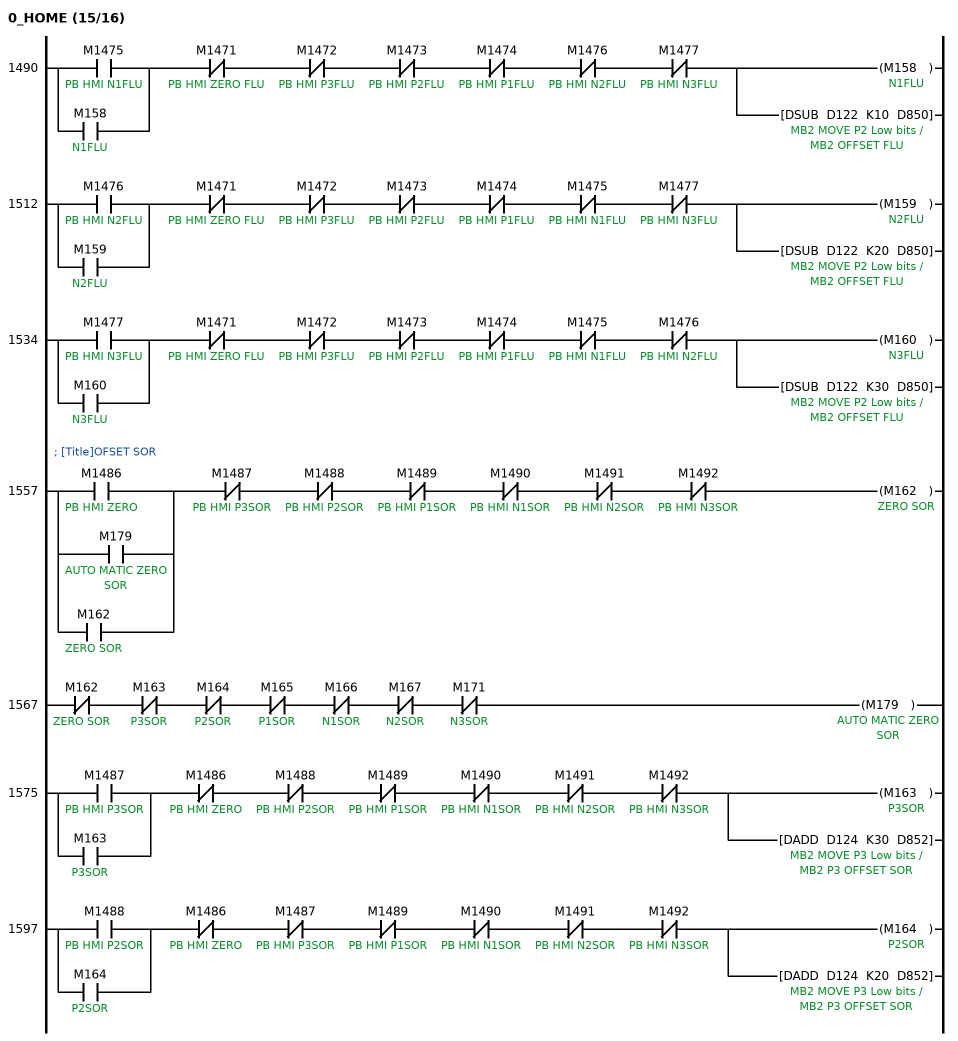
1490  LD      M1475  ; PB HMI N1FLU
      OR      M158  ; N1FLU
      ANI     M1471  ; PB HMI ZERO FLU
      ANI     M1472  ; PB HMI P3FLU
      ANI     M1473  ; PB HMI P2FLU
      ANI     M1474  ; PB HMI P1FLU
      ANI     M1476  ; PB HMI N2FLU
      ANI     M1477  ; PB HMI N3FLU
      OUT     M158  ; N1FLU
      DSUB    D122 K10 D850
1512  LD      M1476  ; PB HMI N2FLU
      OR      M159  ; N2FLU
      ANI     M1471  ; PB HMI ZERO FLU
      ANI     M1472  ; PB HMI P3FLU
      ANI     M1473  ; PB HMI P2FLU
      ANI     M1474  ; PB HMI P1FLU
      ANI     M1475  ; PB HMI N1FLU
      ANI     M1477  ; PB HMI N3FLU
      OUT     M159  ; N2FLU
      DSUB    D122 K20 D850
1534  LD      M1477  ; PB HMI N3FLU
      OR      M160  ; N3FLU
      ANI     M1471  ; PB HMI ZERO FLU
      ANI     M1472  ; PB HMI P3FLU
      ANI     M1473  ; PB HMI P2FLU
      ANI     M1474  ; PB HMI P1FLU
      ANI     M1475  ; PB HMI N1FLU
      ANI     M1476  ; PB HMI N2FLU
      OUT     M160  ; N3FLU
      DSUB    D122 K30 D850
; [Title]OFSET SOR
1557  LD      M1486  ; PB HMI ZERO
      OR      M179  ; AUTO MATIC ZERO SOR
      OR      M162  ; ZERO SOR
      ANI     M1487  ; PB HMI P3SOR
      ANI     M1488  ; PB HMI P2SOR
      ANI     M1489  ; PB HMI P1SOR
      ANI     M1490  ; PB HMI N1SOR
      ANI     M1491  ; PB HMI N2SOR
      ANI     M1492  ; PB HMI N3SOR
      OUT     M162  ; ZERO SOR
1567  LDI     M162  ; ZERO SOR
      ANI     M163  ; P3SOR
      ANI     M164  ; P2SOR
      ANI     M165  ; P1SOR
      ANI     M166  ; N1SOR
      ANI     M167  ; N2SOR
      ANI     M171  ; N3SOR
      OUT     M179  ; AUTO MATIC ZERO SOR
1575  LD      M1487  ; PB HMI P3SOR
      OR      M163  ; P3SOR
      ANI     M1486  ; PB HMI ZERO
      ANI     M1488  ; PB HMI P2SOR
      ANI     M1489  ; PB HMI P1SOR
      ANI     M1490  ; PB HMI N1SOR
      ANI     M1491  ; PB HMI N2SOR
      ANI     M1492  ; PB HMI N3SOR
      OUT     M163  ; P3SOR
      DADD    D124 K30 D852  ; MB2 MOVE P3 Low bits / MB2 P3 OFFSET SOR
1597  LD      M1488  ; PB HMI P2SOR
      OR      M164  ; P2SOR
      ANI     M1486  ; PB HMI ZERO
      ANI     M1487  ; PB HMI P3SOR
      ANI     M1489  ; PB HMI P1SOR
      ANI     M1490  ; PB HMI N1SOR
      ANI     M1491  ; PB HMI N2SOR
      ANI     M1492  ; PB HMI N3SOR
      OUT     M164  ; P2SOR
      DADD    D124 K20 D852
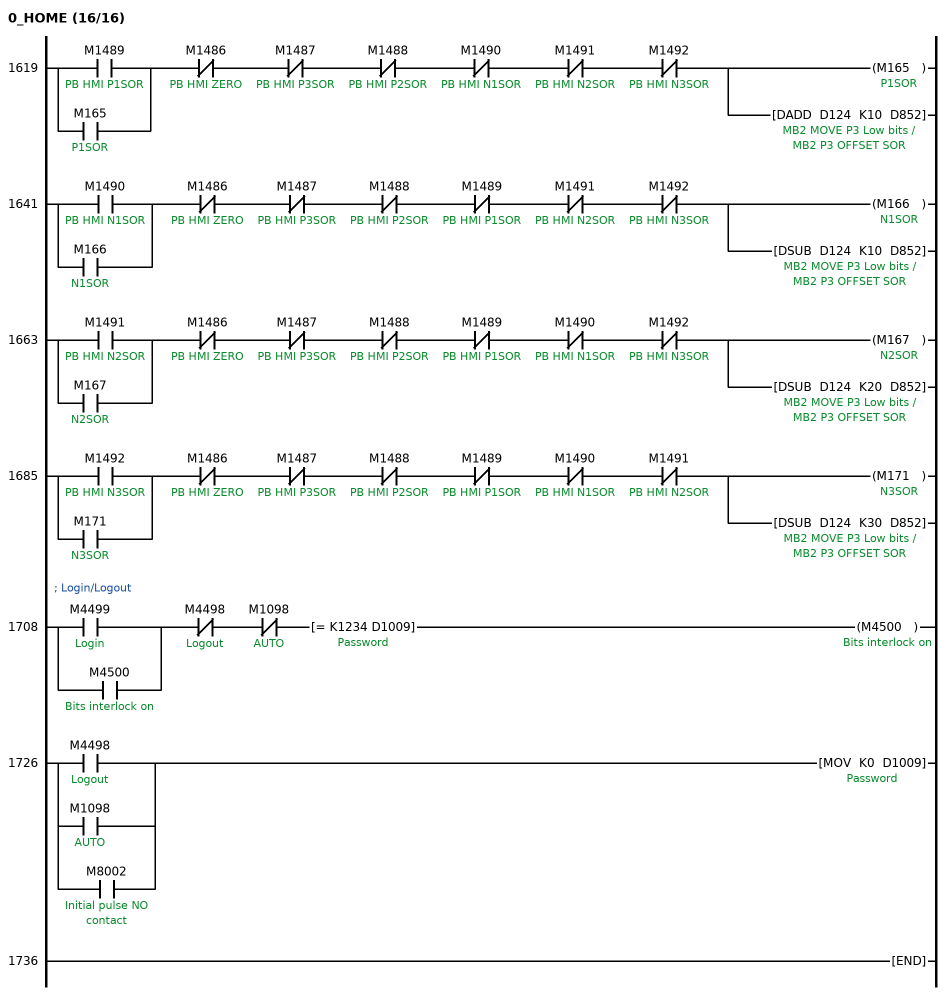
1619  LD      M1489  ; PB HMI P1SOR
      OR      M165  ; P1SOR
      ANI     M1486  ; PB HMI ZERO
      ANI     M1487  ; PB HMI P3SOR
      ANI     M1488  ; PB HMI P2SOR
      ANI     M1490  ; PB HMI N1SOR
      ANI     M1491  ; PB HMI N2SOR
      ANI     M1492  ; PB HMI N3SOR
      OUT     M165  ; P1SOR
      DADD    D124 K10 D852
1641  LD      M1490  ; PB HMI N1SOR
      OR      M166  ; N1SOR
      ANI     M1486  ; PB HMI ZERO
      ANI     M1487  ; PB HMI P3SOR
      ANI     M1488  ; PB HMI P2SOR
      ANI     M1489  ; PB HMI P1SOR
      ANI     M1491  ; PB HMI N2SOR
      ANI     M1492  ; PB HMI N3SOR
      OUT     M166  ; N1SOR
      DSUB    D124 K10 D852
1663  LD      M1491  ; PB HMI N2SOR
      OR      M167  ; N2SOR
      ANI     M1486  ; PB HMI ZERO
      ANI     M1487  ; PB HMI P3SOR
      ANI     M1488  ; PB HMI P2SOR
      ANI     M1489  ; PB HMI P1SOR
      ANI     M1490  ; PB HMI N1SOR
      ANI     M1492  ; PB HMI N3SOR
      OUT     M167  ; N2SOR
      DSUB    D124 K20 D852
1685  LD      M1492  ; PB HMI N3SOR
      OR      M171  ; N3SOR
      ANI     M1486  ; PB HMI ZERO
      ANI     M1487  ; PB HMI P3SOR
      ANI     M1488  ; PB HMI P2SOR
      ANI     M1489  ; PB HMI P1SOR
      ANI     M1490  ; PB HMI N1SOR
      ANI     M1491  ; PB HMI N2SOR
      OUT     M171  ; N3SOR
      DSUB    D124 K30 D852
; Login/Logout
1708  LD      M4499  ; Login
      OR      M4500  ; Bits interlock on
      ANI     M4498  ; Logout
      ANI     M1098  ; AUTO
      AND=    K1234 D1009  ; Password
      OUT     M4500  ; Bits interlock on
1726  LD      M4498  ; Logout
      OR      M1098  ; AUTO
      OR      M8002  ; Initial pulse NO contact
      MOV     K0 D1009
1736  END
END_PROGRAM

PROGRAM 1_MODU_B
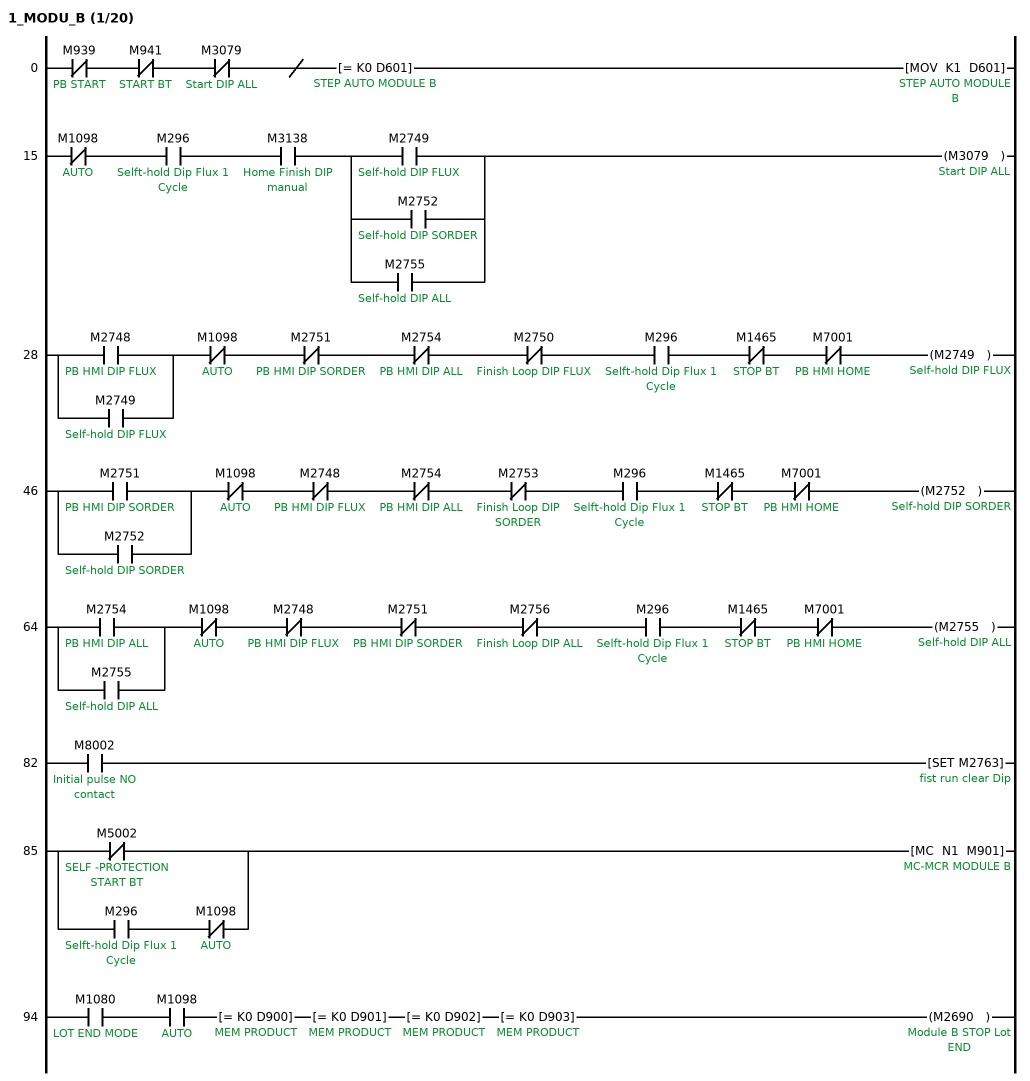
0     LDI     M939  ; PB START
      ANI     M941  ; START BT
      ANI     M3079  ; Start DIP ALL
      INV
      AND=    K0 D601  ; STEP AUTO MODULE B
      MOV     K1 D601
15    LDI     M1098  ; AUTO
      AND     M296  ; Selft-hold Dip Flux 1 Cycle
      AND     M3138  ; Home Finish DIP manual
      LD      M2749  ; Self-hold DIP FLUX
      OR      M2752  ; Self-hold DIP SORDER
      OR      M2755  ; Self-hold DIP ALL
      ANB
      OUT     M3079  ; Start DIP ALL
28    LD      M2748  ; PB HMI DIP FLUX
      OR      M2749  ; Self-hold DIP FLUX
      ANI     M1098  ; AUTO
      ANI     M2751  ; PB HMI DIP SORDER
      ANI     M2754  ; PB HMI DIP ALL
      ANI     M2750  ; Finish Loop DIP FLUX
      AND     M296  ; Selft-hold Dip Flux 1 Cycle
      ANI     M1465  ; STOP BT
      ANI     M7001  ; PB HMI HOME
      OUT     M2749  ; Self-hold DIP FLUX
46    LD      M2751  ; PB HMI DIP SORDER
      OR      M2752  ; Self-hold DIP SORDER
      ANI     M1098  ; AUTO
      ANI     M2748  ; PB HMI DIP FLUX
      ANI     M2754  ; PB HMI DIP ALL
      ANI     M2753  ; Finish Loop DIP SORDER
      AND     M296  ; Selft-hold Dip Flux 1 Cycle
      ANI     M1465  ; STOP BT
      ANI     M7001  ; PB HMI HOME
      OUT     M2752  ; Self-hold DIP SORDER
64    LD      M2754  ; PB HMI DIP ALL
      OR      M2755  ; Self-hold DIP ALL
      ANI     M1098  ; AUTO
      ANI     M2748  ; PB HMI DIP FLUX
      ANI     M2751  ; PB HMI DIP SORDER
      ANI     M2756  ; Finish Loop DIP ALL
      AND     M296  ; Selft-hold Dip Flux 1 Cycle
      ANI     M1465  ; STOP BT
      ANI     M7001  ; PB HMI HOME
      OUT     M2755  ; Self-hold DIP ALL
82    LD      M8002  ; Initial pulse NO contact
      SET     M2763  ; fist run clear Dip
85    LDI     M5002  ; SELF -PROTECTION START BT
      LD      M296  ; Selft-hold Dip Flux 1 Cycle
      ANI     M1098  ; AUTO
      ORB
      MC      N1 M901  ; MC-MCR MODULE B
94    LD      M1080  ; LOT END MODE
      AND     M1098  ; AUTO
      AND=    K0 D900  ; MEM PRODUCT
      AND=    K0 D901  ; MEM PRODUCT
      AND=    K0 D902  ; MEM PRODUCT
      AND=    K0 D903  ; MEM PRODUCT
      OUT     M2690  ; Module B STOP Lot END
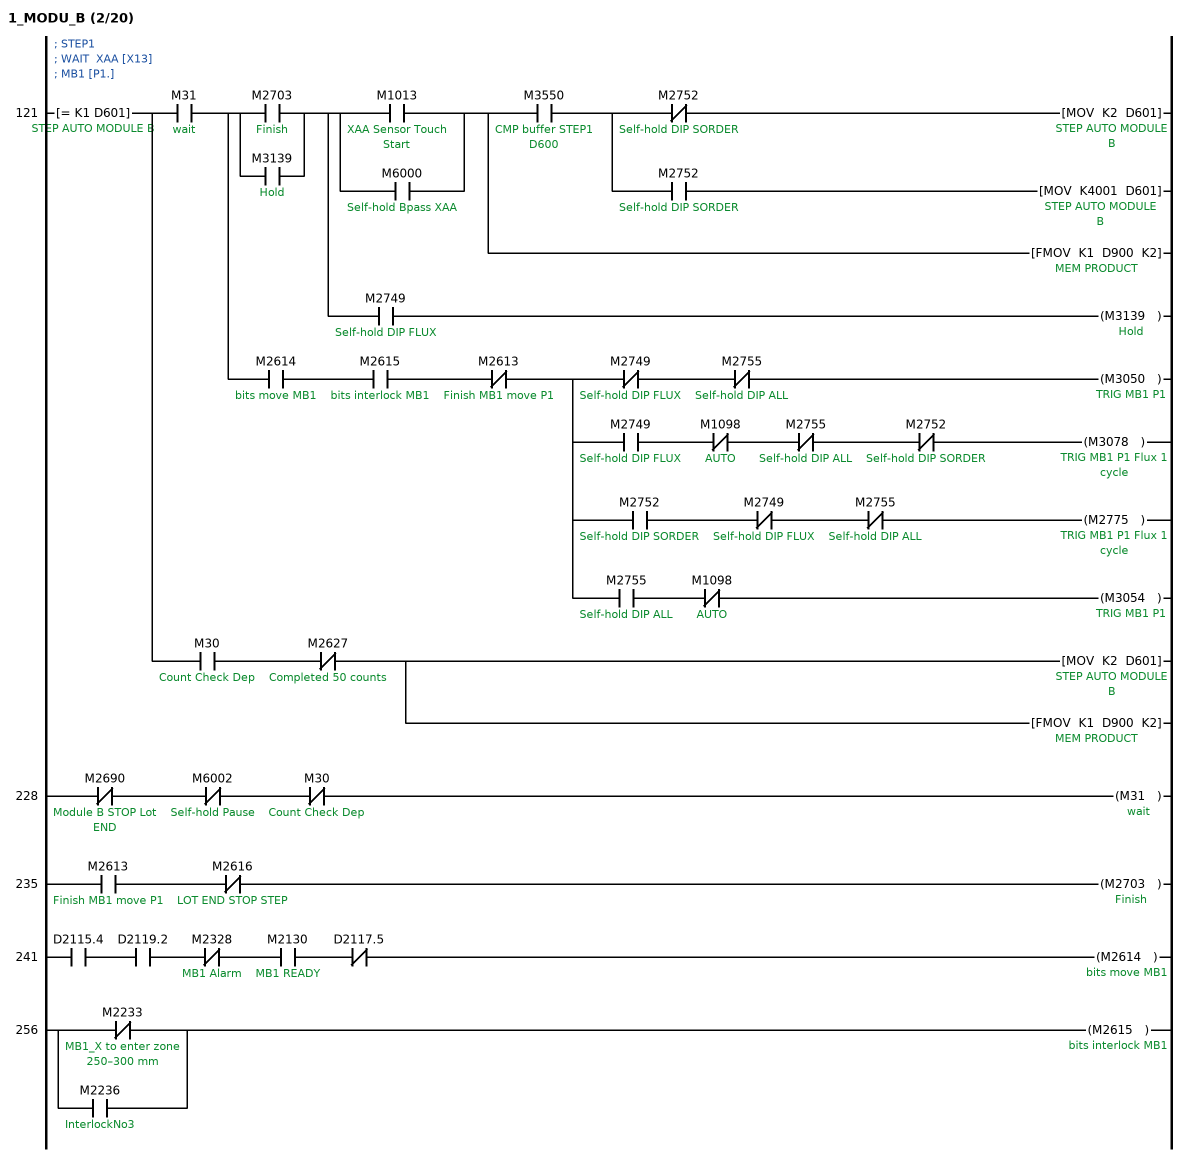
; STEP1
; WAIT  XAA [X13]
; MB1 [P1.]
121   LD=     K1 D601  ; STEP AUTO MODULE B
      MPS
      AND     M31  ; wait
      MPS
      LD      M2703  ; Finish
      OR      M3139  ; Hold
      ANB
      MPS
      LD      M1013  ; XAA Sensor Touch Start
      OR      M6000  ; Self-hold Bpass XAA
      ANB
      MPS
      AND     M3550  ; CMP buffer STEP1 D600
      MPS
      ANI     M2752  ; Self-hold DIP SORDER
      MOV     K2 D601
      MPP
      AND     M2752  ; Self-hold DIP SORDER
      MOV     K4001 D601
      MPP
      FMOV    K1 D900 K2
      MPP
      AND     M2749  ; Self-hold DIP FLUX
      OUT     M3139  ; Hold
      MPP
      AND     M2614  ; bits move MB1
      AND     M2615  ; bits interlock MB1
      ANI     M2613  ; Finish MB1 move P1
      MPS
      ANI     M2749  ; Self-hold DIP FLUX
      ANI     M2755  ; Self-hold DIP ALL
      OUT     M3050  ; TRIG MB1 P1
        [note] TRIG MB1 P1
      MRD
      AND     M2749  ; Self-hold DIP FLUX
      ANI     M1098  ; AUTO
      ANI     M2755  ; Self-hold DIP ALL
      ANI     M2752  ; Self-hold DIP SORDER
      OUT     M3078  ; TRIG MB1 P1 Flux 1 cycle
      MRD
      AND     M2752  ; Self-hold DIP SORDER
      ANI     M2749  ; Self-hold DIP FLUX
      ANI     M2755  ; Self-hold DIP ALL
      OUT     M2775  ; TRIG MB1 P1 Flux 1 cycle
      MPP
      AND     M2755  ; Self-hold DIP ALL
      ANI     M1098  ; AUTO
      OUT     M3054  ; TRIG MB1 P1
      MPP
      AND     M30  ; Count Check Dep
      ANI     M2627  ; Completed 50 counts
      MOV     K2 D601
      FMOV    K1 D900 K2
228   LDI     M2690  ; Module B STOP Lot END
      ANI     M6002  ; Self-hold Pause
      ANI     M30  ; Count Check Dep
      OUT     M31  ; wait
235   LD      M2613  ; Finish MB1 move P1
      ANI     M2616  ; LOT END STOP STEP
      OUT     M2703  ; Finish
241   LD      D2115.4
      AND     D2119.2
      ANI     M2328  ; MB1 Alarm
      AND     M2130  ; MB1 READY
      ANI     D2117.5
      OUT     M2614  ; bits move MB1
256   LDI     M2233  ; MB1_X to enter zone 250–300 mm
      OR      M2236  ; InterlockNo3
      OUT     M2615  ; bits interlock MB1
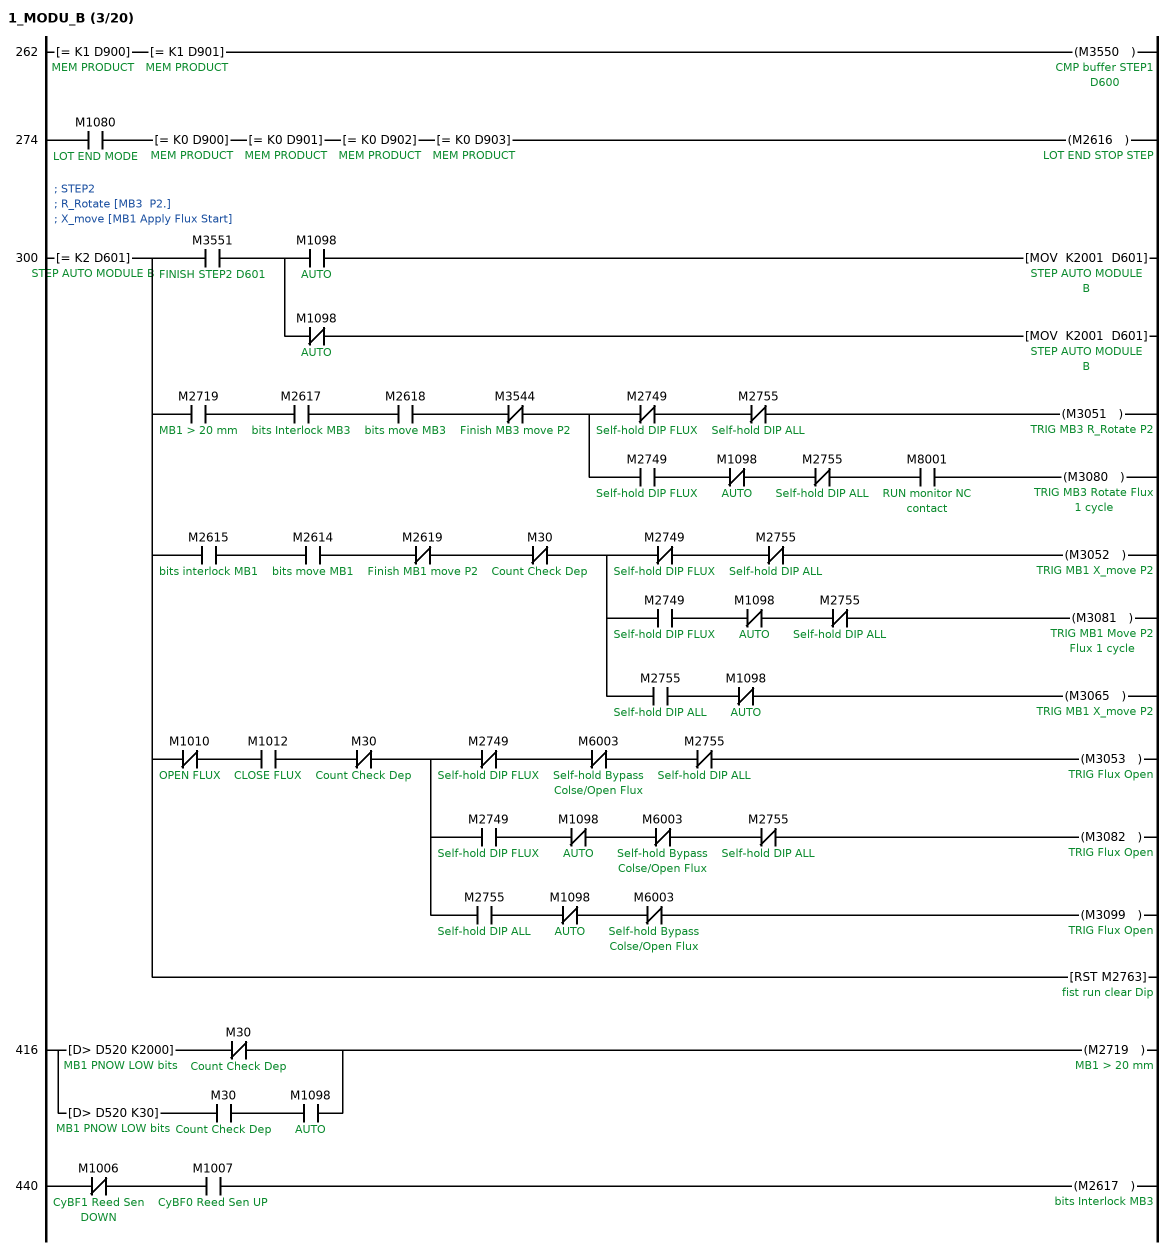
262   LD=     K1 D900  ; MEM PRODUCT
      AND=    K1 D901  ; MEM PRODUCT
      OUT     M3550  ; CMP buffer STEP1 D600
274   LD      M1080  ; LOT END MODE
      AND=    K0 D900  ; MEM PRODUCT
      AND=    K0 D901  ; MEM PRODUCT
      AND=    K0 D902  ; MEM PRODUCT
      AND=    K0 D903  ; MEM PRODUCT
      OUT     M2616  ; LOT END STOP STEP
; STEP2
; R_Rotate [MB3  P2.]
; X_move [MB1 Apply Flux Start]
300   LD=     K2 D601  ; STEP AUTO MODULE B
      MPS
      AND     M3551  ; FINISH STEP2 D601
      MPS
      AND     M1098  ; AUTO
      MOV     K2001 D601
      MPP
      ANI     M1098  ; AUTO
      MOV     K2001 D601
      MRD
      AND     M2719  ; MB1 > 20 mm
      AND     M2617  ; bits Interlock MB3
      AND     M2618  ; bits move MB3
      ANI     M3544  ; Finish MB3 move P2
      MPS
      ANI     M2749  ; Self-hold DIP FLUX
      ANI     M2755  ; Self-hold DIP ALL
      OUT     M3051  ; TRIG MB3 R_Rotate P2
        [note] TRIG MB3 R_Rotate P2
      MPP
      AND     M2749  ; Self-hold DIP FLUX
      ANI     M1098  ; AUTO
      ANI     M2755  ; Self-hold DIP ALL
      AND     M8001  ; RUN monitor NC contact
      OUT     M3080  ; TRIG MB3 Rotate Flux 1 cycle
      MRD
      AND     M2615  ; bits interlock MB1
      AND     M2614  ; bits move MB1
      ANI     M2619  ; Finish MB1 move P2
      ANI     M30  ; Count Check Dep
      MPS
      ANI     M2749  ; Self-hold DIP FLUX
      ANI     M2755  ; Self-hold DIP ALL
      OUT     M3052  ; TRIG MB1 X_move P2
        [note] TRIG MB1 X_move P2
      MRD
      AND     M2749  ; Self-hold DIP FLUX
      ANI     M1098  ; AUTO
      ANI     M2755  ; Self-hold DIP ALL
      OUT     M3081  ; TRIG MB1 Move P2 Flux 1 cycle
      MPP
      AND     M2755  ; Self-hold DIP ALL
      ANI     M1098  ; AUTO
      OUT     M3065  ; TRIG MB1 X_move P2
      MRD
      ANI     M1010  ; OPEN FLUX
      AND     M1012  ; CLOSE FLUX
      ANI     M30  ; Count Check Dep
      MPS
      ANI     M2749  ; Self-hold DIP FLUX
      ANI     M6003  ; Self-hold Bypass Colse/Open Flux
      ANI     M2755  ; Self-hold DIP ALL
      OUT     M3053  ; TRIG Flux Open
        [note] TRIG Flux Open
      MRD
      AND     M2749  ; Self-hold DIP FLUX
      ANI     M1098  ; AUTO
      ANI     M6003  ; Self-hold Bypass Colse/Open Flux
      ANI     M2755  ; Self-hold DIP ALL
      OUT     M3082  ; TRIG Flux Open
      MPP
      AND     M2755  ; Self-hold DIP ALL
      ANI     M1098  ; AUTO
      ANI     M6003  ; Self-hold Bypass Colse/Open Flux
      OUT     M3099  ; TRIG Flux Open
      MPP
      RST     M2763  ; fist run clear Dip
416   LDD>    D520 K2000  ; MB1 PNOW LOW bits
      ANI     M30  ; Count Check Dep
      LDD>    D520 K30  ; MB1 PNOW LOW bits
      AND     M30  ; Count Check Dep
      AND     M1098  ; AUTO
      ORB
      OUT     M2719  ; MB1 > 20 mm
440   LDI     M1006  ; CyBF1 Reed Sen DOWN
      AND     M1007  ; CyBF0 Reed Sen UP
      OUT     M2617  ; bits Interlock MB3
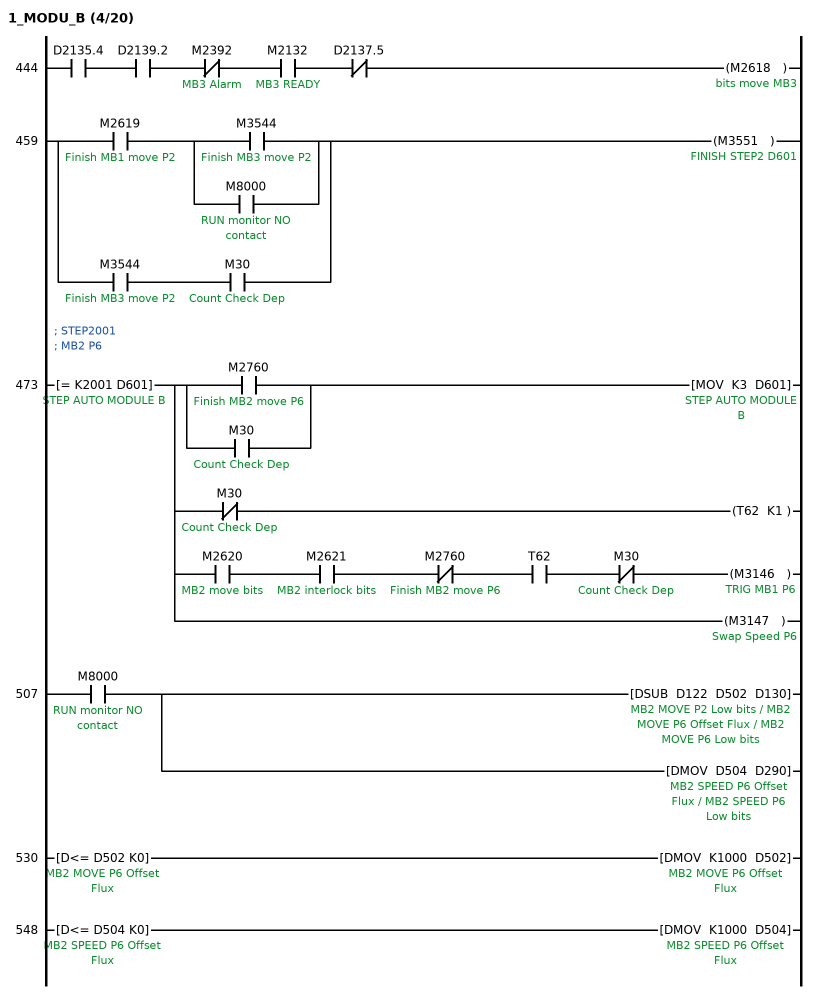
444   LD      D2135.4
      AND     D2139.2
      ANI     M2392  ; MB3 Alarm
      AND     M2132  ; MB3 READY
      ANI     D2137.5
      OUT     M2618  ; bits move MB3
459   LD      M2619  ; Finish MB1 move P2
      LD      M3544  ; Finish MB3 move P2
      OR      M8000  ; RUN monitor NO contact
      ANB
      LD      M3544  ; Finish MB3 move P2
      AND     M30  ; Count Check Dep
      ORB
      OUT     M3551  ; FINISH STEP2 D601
; STEP2001
; MB2 P6
473   LD=     K2001 D601  ; STEP AUTO MODULE B
      MPS
      LD      M2760  ; Finish MB2 move P6
      OR      M30  ; Count Check Dep
      ANB
      MOV     K3 D601
      MRD
      ANI     M30  ; Count Check Dep
      OUT     T62 K1
      MRD
      AND     M2620  ; MB2 move bits
      AND     M2621  ; MB2 interlock bits
      ANI     M2760  ; Finish MB2 move P6
      AND     T62
      ANI     M30  ; Count Check Dep
      OUT     M3146  ; TRIG MB1 P6
      MPP
      OUT     M3147  ; Swap Speed P6
507   LD      M8000  ; RUN monitor NO contact
      DSUB    D122 D502 D130  ; MB2 MOVE P2 Low bits / MB2 MOVE P6 Offset Flux / MB2 MOVE P6 Low bits
      DMOV    D504 D290  ; MB2 SPEED P6 Offset Flux / MB2 SPEED P6 Low bits
530   LDD<=   D502 K0  ; MB2 MOVE P6 Offset Flux
      DMOV    K1000 D502
548   LDD<=   D504 K0  ; MB2 SPEED P6 Offset Flux
      DMOV    K1000 D504
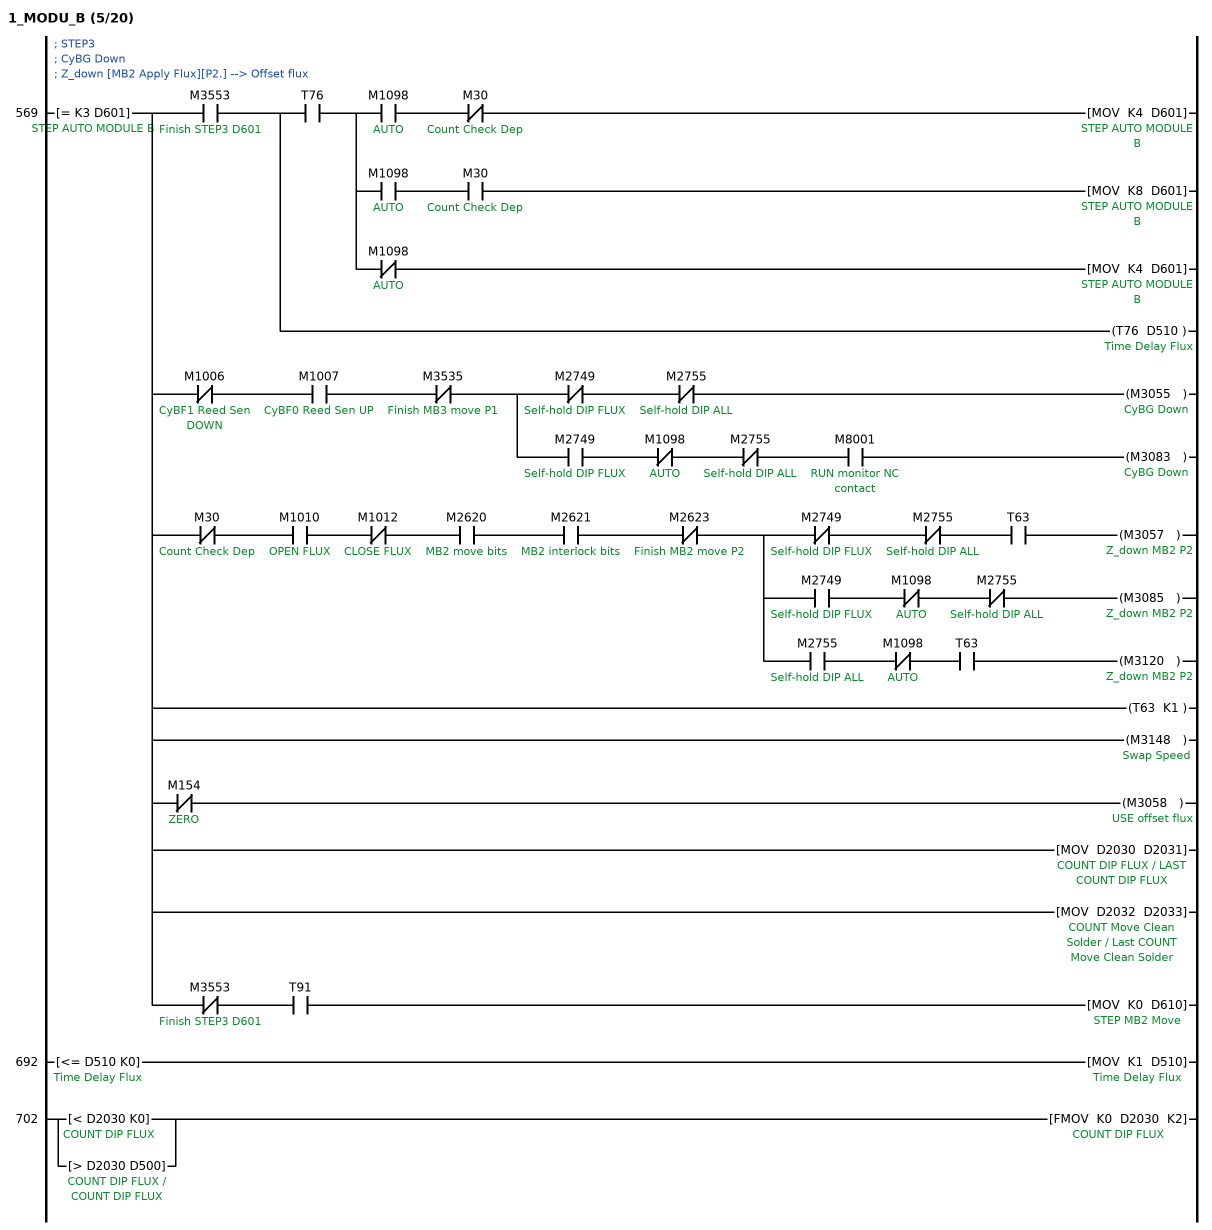
; STEP3
; CyBG Down
; Z_down [MB2 Apply Flux][P2.] --> Offset flux
569   LD=     K3 D601  ; STEP AUTO MODULE B
      MPS
      AND     M3553  ; Finish STEP3 D601
      MPS
      AND     T76
      MPS
      AND     M1098  ; AUTO
      ANI     M30  ; Count Check Dep
      MOV     K4 D601
      MRD
      AND     M1098  ; AUTO
      AND     M30  ; Count Check Dep
      MOV     K8 D601
      MPP
      ANI     M1098  ; AUTO
      MOV     K4 D601
      MPP
      OUT     T76 D510  ; Time Delay Flux
      MRD
      ANI     M1006  ; CyBF1 Reed Sen DOWN
      AND     M1007  ; CyBF0 Reed Sen UP
      ANI     M3535  ; Finish MB3 move P1
      MPS
      ANI     M2749  ; Self-hold DIP FLUX
      ANI     M2755  ; Self-hold DIP ALL
      OUT     M3055  ; CyBG Down
        [note] CyBG Down
      MPP
      AND     M2749  ; Self-hold DIP FLUX
      ANI     M1098  ; AUTO
      ANI     M2755  ; Self-hold DIP ALL
      AND     M8001  ; RUN monitor NC contact
      OUT     M3083  ; CyBG Down
      MRD
      ANI     M30  ; Count Check Dep
      AND     M1010  ; OPEN FLUX
      ANI     M1012  ; CLOSE FLUX
      AND     M2620  ; MB2 move bits
      AND     M2621  ; MB2 interlock bits
      ANI     M2623  ; Finish MB2 move P2
      MPS
      ANI     M2749  ; Self-hold DIP FLUX
      ANI     M2755  ; Self-hold DIP ALL
      AND     T63
      OUT     M3057  ; Z_down MB2 P2
        [note] TRIG Z_down MB2 P2
      MRD
      AND     M2749  ; Self-hold DIP FLUX
      ANI     M1098  ; AUTO
      ANI     M2755  ; Self-hold DIP ALL
      OUT     M3085  ; Z_down MB2 P2
      MPP
      AND     M2755  ; Self-hold DIP ALL
      ANI     M1098  ; AUTO
      AND     T63
      OUT     M3120  ; Z_down MB2 P2
      MPP
      OUT     T63 K1
      OUT     M3148  ; Swap Speed
      MPS
      ANI     M154  ; ZERO
      OUT     M3058  ; USE offset flux
        [note] USE OFFSET FLUX
      MPP
      MOV     D2030 D2031  ; COUNT DIP FLUX / LAST COUNT DIP FLUX
      MOV     D2032 D2033  ; COUNT Move Clean Solder / Last COUNT Move Clean Solder
      ANI     M3553  ; Finish STEP3 D601
      AND     T91
      MOV     K0 D610  ; STEP MB2 Move
692   LD<=    D510 K0  ; Time Delay Flux
      MOV     K1 D510
702   LD<     D2030 K0  ; COUNT DIP FLUX
      OR>     D2030 D500  ; COUNT DIP FLUX / COUNT DIP FLUX
      FMOV    K0 D2030 K2
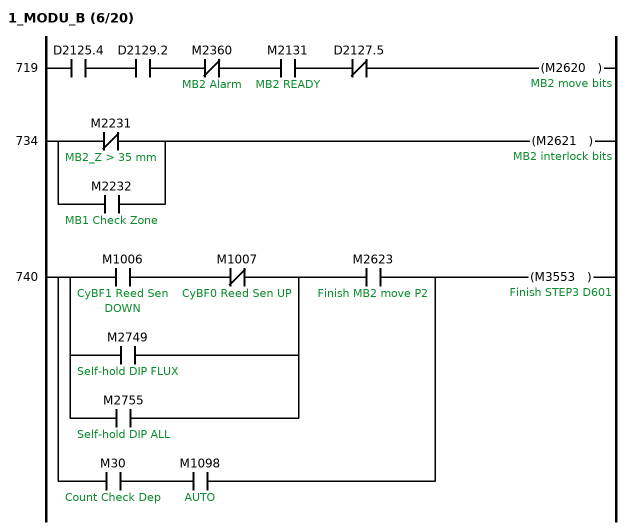
719   LD      D2125.4
      AND     D2129.2
      ANI     M2360  ; MB2 Alarm
      AND     M2131  ; MB2 READY
      ANI     D2127.5
      OUT     M2620  ; MB2 move bits
734   LDI     M2231  ; MB2_Z > 35 mm
      OR      M2232  ; MB1 Check Zone
      OUT     M2621  ; MB2 interlock bits
740   LD      M1006  ; CyBF1 Reed Sen DOWN
      ANI     M1007  ; CyBF0 Reed Sen UP
      OR      M2749  ; Self-hold DIP FLUX
      OR      M2755  ; Self-hold DIP ALL
      AND     M2623  ; Finish MB2 move P2
      LD      M30  ; Count Check Dep
      AND     M1098  ; AUTO
      ORB
      OUT     M3553  ; Finish STEP3 D601
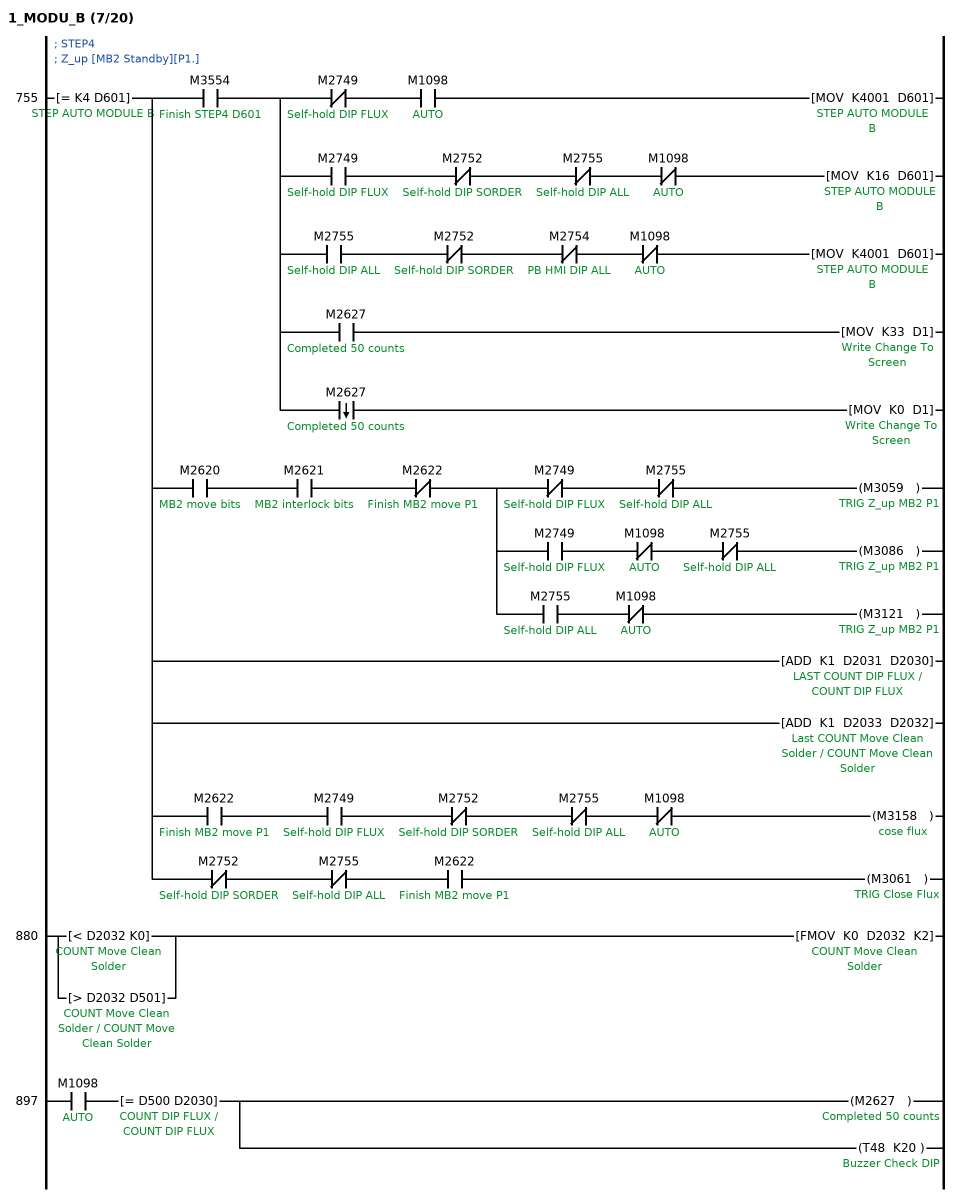
; STEP4
; Z_up [MB2 Standby][P1.]
755   LD=     K4 D601  ; STEP AUTO MODULE B
      MPS
      AND     M3554  ; Finish STEP4 D601
      MPS
      ANI     M2749  ; Self-hold DIP FLUX
      AND     M1098  ; AUTO
      MOV     K4001 D601
      MRD
      AND     M2749  ; Self-hold DIP FLUX
      ANI     M2752  ; Self-hold DIP SORDER
      ANI     M2755  ; Self-hold DIP ALL
      ANI     M1098  ; AUTO
      MOV     K16 D601
      MRD
      AND     M2755  ; Self-hold DIP ALL
      ANI     M2752  ; Self-hold DIP SORDER
      ANI     M2754  ; PB HMI DIP ALL
      ANI     M1098  ; AUTO
      MOV     K4001 D601
      MRD
      AND     M2627  ; Completed 50 counts
      MOV     K33 D1  ; Write Change To Screen
      MPP
      ANDF    M2627  ; Completed 50 counts
      MOV     K0 D1
      MRD
      AND     M2620  ; MB2 move bits
      AND     M2621  ; MB2 interlock bits
      ANI     M2622  ; Finish MB2 move P1
      MPS
      ANI     M2749  ; Self-hold DIP FLUX
      ANI     M2755  ; Self-hold DIP ALL
      OUT     M3059  ; TRIG Z_up MB2 P1
        [note] TRIG Z_up MB2 P1
      MRD
      AND     M2749  ; Self-hold DIP FLUX
      ANI     M1098  ; AUTO
      ANI     M2755  ; Self-hold DIP ALL
      OUT     M3086  ; TRIG Z_up MB2 P1
      MPP
      AND     M2755  ; Self-hold DIP ALL
      ANI     M1098  ; AUTO
      OUT     M3121  ; TRIG Z_up MB2 P1
      MPP
      ADD     K1 D2031 D2030
      ADD     K1 D2033 D2032
      MPS
      AND     M2622  ; Finish MB2 move P1
      AND     M2749  ; Self-hold DIP FLUX
      ANI     M2752  ; Self-hold DIP SORDER
      ANI     M2755  ; Self-hold DIP ALL
      ANI     M1098  ; AUTO
      OUT     M3158  ; cose flux
      MPP
      ANI     M2752  ; Self-hold DIP SORDER
      ANI     M2755  ; Self-hold DIP ALL
      AND     M2622  ; Finish MB2 move P1
      OUT     M3061  ; TRIG Close Flux
        [note] TRIG Close Flux
880   LD<     D2032 K0  ; COUNT Move Clean Solder
      OR>     D2032 D501  ; COUNT Move Clean Solder / COUNT Move Clean Solder
      FMOV    K0 D2032 K2
897   LD      M1098  ; AUTO
      AND=    D500 D2030  ; COUNT DIP FLUX / COUNT DIP FLUX
      OUT     M2627  ; Completed 50 counts
      OUT     T48 K20  ; Buzzer Check DIP
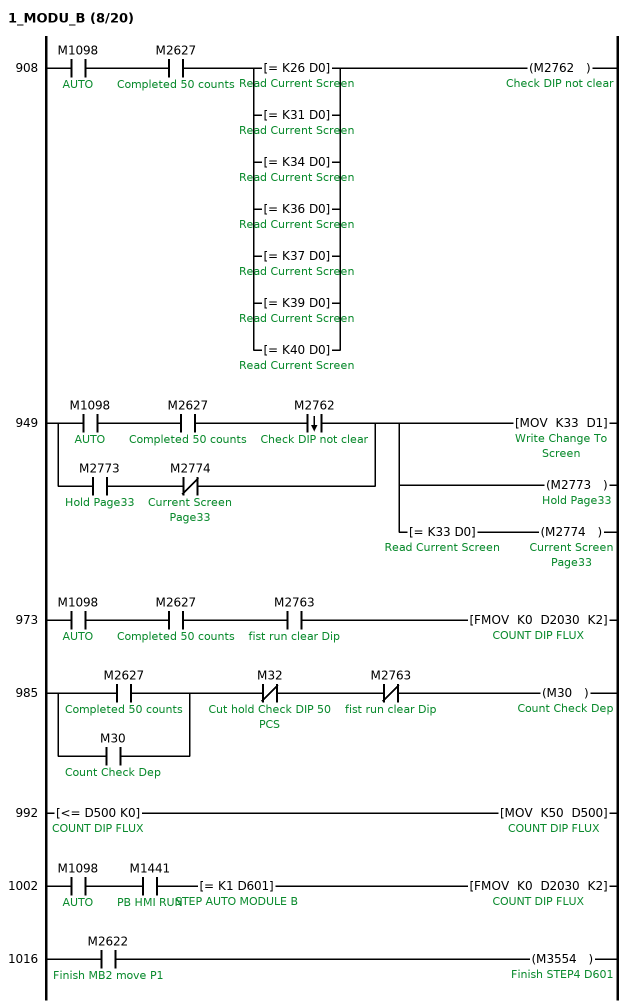
908   LD      M1098  ; AUTO
      AND     M2627  ; Completed 50 counts
      LD=     K26 D0  ; Read Current Screen
      OR=     K31 D0  ; Read Current Screen
      OR=     K34 D0  ; Read Current Screen
      OR=     K36 D0  ; Read Current Screen
      OR=     K37 D0  ; Read Current Screen
      OR=     K39 D0  ; Read Current Screen
      OR=     K40 D0  ; Read Current Screen
      ANB
      OUT     M2762  ; Check DIP not clear
949   LD      M1098  ; AUTO
      AND     M2627  ; Completed 50 counts
      ANDF    M2762  ; Check DIP not clear
      LD      M2773  ; Hold Page33
      ANI     M2774  ; Current Screen Page33
      ORB
      MOV     K33 D1
      OUT     M2773  ; Hold Page33
      AND=    K33 D0  ; Read Current Screen
      OUT     M2774  ; Current Screen Page33
973   LD      M1098  ; AUTO
      AND     M2627  ; Completed 50 counts
      AND     M2763  ; fist run clear Dip
      FMOV    K0 D2030 K2
985   LD      M2627  ; Completed 50 counts
      OR      M30  ; Count Check Dep
      ANI     M32  ; Cut hold Check DIP 50 PCS
      ANI     M2763  ; fist run clear Dip
      OUT     M30  ; Count Check Dep
992   LD<=    D500 K0  ; COUNT DIP FLUX
      MOV     K50 D500
1002  LD      M1098  ; AUTO
      AND     M1441  ; PB HMI RUN
      AND=    K1 D601  ; STEP AUTO MODULE B
      FMOV    K0 D2030 K2
1016  LD      M2622  ; Finish MB2 move P1
      OUT     M3554  ; Finish STEP4 D601
